        (* End of MultiPortSwitch: '<S729>/Multiport Switch' *)
        

        (* Sum: '<S308>/Add' incorporates:
         *  Constant: '<S304>/Constant'
         *  Product: '<S308>/Product' *)
        rtb_Add_d := USINT_TO_REAL(C_Actia_Batt2_ADS_8[5]) * 5.0;
        (* Sum: '<S547>/Add' incorporates:
         *  ArithShift: '<S546>/Shift Arithmetic'
         *  DataTypeConversion: '<S546>/Data Type Conversion'
         *  Sum: '<S546>/Add' *)
        rtb_Add_ci := DINT_TO_REAL(DWORD_TO_DINT(SHL(DINT_TO_DWORD(USINT_TO_DINT(C_LB_Batt2_InsulationMonitor_Msg[1])), 8)) + USINT_TO_DINT(C_LB_Batt2_InsulationMonitor_Msg[0]));
        (* Switch: '<S547>/Switch' incorporates:
         *  Constant: '<S543>/Constant4' *)

        IF C_LB_Batt2_InsulationMonitor_Timeout THEN 
            rtb_Add_ci := 0.0;
        END_IF;

        (* End of Switch: '<S547>/Switch' *)
        

        (* Sum: '<S730>/Subtract' incorporates:
         *  Constant: '<S730>/Constant4'
         *  Gain: '<S730>/mV to V' *)
        rtb_Add_ci := (0.001 * rtb_Add_ci) - 2.48;
        (* MultiPortSwitch: '<S727>/Multiport Switch' incorporates:
         *  Abs: '<S730>/Abs'
         *  Constant: '<S727>/Constant'
         *  Constant: '<S730>/Constant1'
         *  Constant: '<S730>/Constant2'
         *  Product: '<S730>/Divide'
         *  Product: '<S730>/Product'
         *  Sum: '<S730>/Subtract1' *)

        CASE TRUNC(rtb_BattSelect) OF
            1: 
                (* Switch: '<S308>/Switch' incorporates:
                 *  Constant: '<S304>/Constant3'
                 *  Constant: '<S304>/SafeValue_NA '
                 *  RelationalOperator: '<S308>/GreaterThan'
                 *  Switch: '<S308>/Switch1' *)

                IF C_Actia_Batt2_ADS_8_Timeout THEN 
                    rtb_Add_d := 0.0;
                ELSIF rtb_Add_d > 0.0 THEN 
                    (* Switch: '<S308>/Switch1' incorporates:
                     *  Constant: '<S304>/SafeValue_Error' *)
                    rtb_Add_d := 0.0;
                END_IF;

                (* End of Switch: '<S308>/Switch' *)
            2: 
                rtb_Add_d := ((rtb_Add_ic * 10.0) / ABS(rtb_Add_ci)) - 2000.0;
            3: 
                rtb_Add_d := 0.0;
            ELSE
                rtb_Add_d := 0.0;
        END_CASE;

        (* End of MultiPortSwitch: '<S727>/Multiport Switch' *)
        

        (* Sum: '<S369>/Add' incorporates:
         *  Constant: '<S365>/Constant'
         *  Product: '<S369>/Product' *)
        rtb_Add_ky := USINT_TO_REAL(C_Actia_Batt3_ADS_8[5]) * 5.0;
        (* Sum: '<S627>/Add' incorporates:
         *  ArithShift: '<S626>/Shift Arithmetic'
         *  DataTypeConversion: '<S626>/Data Type Conversion'
         *  Sum: '<S626>/Add' *)
        rtb_Add_ci := DINT_TO_REAL(DWORD_TO_DINT(SHL(DINT_TO_DWORD(USINT_TO_DINT(C_LB_Batt3_InsulationMonitor_Msg[1])), 8)) + USINT_TO_DINT(C_LB_Batt3_InsulationMonitor_Msg[0]));
        (* Switch: '<S627>/Switch' incorporates:
         *  Constant: '<S623>/Constant4' *)

        IF C_LB_Batt3_InsulationMonitor_Timeout THEN 
            rtb_Add_ci := 0.0;
        END_IF;

        (* End of Switch: '<S627>/Switch' *)
        

        (* Sum: '<S731>/Subtract' incorporates:
         *  Constant: '<S731>/Constant4'
         *  Gain: '<S731>/mV to V' *)
        rtb_Add_ci := (0.001 * rtb_Add_ci) - 2.48;
        (* MultiPortSwitch: '<S728>/Multiport Switch' incorporates:
         *  Abs: '<S731>/Abs'
         *  Constant: '<S728>/Constant'
         *  Constant: '<S731>/Constant1'
         *  Constant: '<S731>/Constant2'
         *  Product: '<S731>/Divide'
         *  Product: '<S731>/Product'
         *  Sum: '<S731>/Subtract1' *)

        CASE TRUNC(rtb_BattSelect_i) OF
            1: 
                (* Switch: '<S369>/Switch' incorporates:
                 *  Constant: '<S365>/Constant3'
                 *  Constant: '<S365>/SafeValue_NA '
                 *  RelationalOperator: '<S369>/GreaterThan'
                 *  Switch: '<S369>/Switch1' *)

                IF C_Actia_Batt3_ADS_8_Timeout THEN 
                    rtb_Add_ky := 0.0;
                ELSIF rtb_Add_ky > 0.0 THEN 
                    (* Switch: '<S369>/Switch1' incorporates:
                     *  Constant: '<S365>/SafeValue_Error' *)
                    rtb_Add_ky := 0.0;
                END_IF;

                (* End of Switch: '<S369>/Switch' *)
            2: 
                rtb_Add_ky := ((rtb_Add_en * 10.0) / ABS(rtb_Add_ci)) - 2000.0;
            3: 
                rtb_Add_ky := 0.0;
            ELSE
                rtb_Add_ky := 0.0;
        END_CASE;

        (* End of MultiPortSwitch: '<S728>/Multiport Switch' *)
        

        (* Sum: '<S469>/Add' incorporates:
         *  ArithShift: '<S468>/Shift Arithmetic'
         *  DataTypeConversion: '<S468>/Data Type Conversion'
         *  Sum: '<S468>/Add' *)
        rtb_Add_ci := DINT_TO_REAL(DWORD_TO_DINT(SHL(DINT_TO_DWORD(USINT_TO_DINT(C_LB_Batt1_InsulationMonitor_Msg[3])), 8)) + USINT_TO_DINT(C_LB_Batt1_InsulationMonitor_Msg[2]));
        (* Switch: '<S469>/Switch' incorporates:
         *  Constant: '<S464>/Constant4' *)

        IF C_LB_Batt1_InsulationMonitor_Timeout THEN 
            rtb_Add_ci := 0.0;
        END_IF;

        (* End of Switch: '<S469>/Switch' *)
        

        (* Sum: '<S732>/Subtract3' incorporates:
         *  Abs: '<S732>/Abs1'
         *  Constant: '<S732>/Constant5'
         *  Constant: '<S732>/Constant6'
         *  Constant: '<S732>/Constant7'
         *  Gain: '<S732>/mV to V1'
         *  Product: '<S732>/Divide1'
         *  Product: '<S732>/Product1'
         *  Sum: '<S732>/Subtract2' *)
        rtb_Add_psl := ((rtb_Add_psl * 10.0) / ABS((0.001 * rtb_Add_ci) - 2.48)) - 2000.0;
        (* Sum: '<S549>/Add' incorporates:
         *  ArithShift: '<S548>/Shift Arithmetic'
         *  DataTypeConversion: '<S548>/Data Type Conversion'
         *  Sum: '<S548>/Add' *)
        rtb_Add_ci := DINT_TO_REAL(DWORD_TO_DINT(SHL(DINT_TO_DWORD(USINT_TO_DINT(C_LB_Batt2_InsulationMonitor_Msg[3])), 8)) + USINT_TO_DINT(C_LB_Batt2_InsulationMonitor_Msg[2]));
        (* Switch: '<S549>/Switch' incorporates:
         *  Constant: '<S544>/Constant4' *)

        IF C_LB_Batt2_InsulationMonitor_Timeout THEN 
            rtb_Add_ci := 0.0;
        END_IF;

        (* End of Switch: '<S549>/Switch' *)
        

        (* Sum: '<S730>/Subtract3' incorporates:
         *  Abs: '<S730>/Abs1'
         *  Constant: '<S730>/Constant5'
         *  Constant: '<S730>/Constant6'
         *  Constant: '<S730>/Constant7'
         *  Gain: '<S730>/mV to V1'
         *  Product: '<S730>/Divide1'
         *  Product: '<S730>/Product1'
         *  Sum: '<S730>/Subtract2' *)
        rtb_Add_ic := ((rtb_Add_ic * 10.0) / ABS((0.001 * rtb_Add_ci) - 2.48)) - 2000.0;
        (* Sum: '<S629>/Add' incorporates:
         *  ArithShift: '<S628>/Shift Arithmetic'
         *  DataTypeConversion: '<S628>/Data Type Conversion'
         *  Sum: '<S628>/Add' *)
        rtb_Add_ci := DINT_TO_REAL(DWORD_TO_DINT(SHL(DINT_TO_DWORD(USINT_TO_DINT(C_LB_Batt3_InsulationMonitor_Msg[3])), 8)) + USINT_TO_DINT(C_LB_Batt3_InsulationMonitor_Msg[2]));
        (* Switch: '<S629>/Switch' incorporates:
         *  Constant: '<S624>/Constant4' *)

        IF C_LB_Batt3_InsulationMonitor_Timeout THEN 
            rtb_Add_ci := 0.0;
        END_IF;

        (* End of Switch: '<S629>/Switch' *)
        

        (* Sum: '<S731>/Subtract3' incorporates:
         *  Abs: '<S731>/Abs1'
         *  Constant: '<S731>/Constant5'
         *  Constant: '<S731>/Constant6'
         *  Constant: '<S731>/Constant7'
         *  Gain: '<S731>/mV to V1'
         *  Product: '<S731>/Divide1'
         *  Product: '<S731>/Product1'
         *  Sum: '<S731>/Subtract2' *)
        rtb_Add_en := ((rtb_Add_en * 10.0) / ABS((0.001 * rtb_Add_ci) - 2.48)) - 2000.0;
        (* Sum: '<S259>/Add' incorporates:
         *  Product: '<S259>/Product' *)
        rtb_Switch_a := USINT_TO_REAL(C_Actia_Batt1_ADS_1[7]);
        (* MultiPortSwitch: '<S726>/Multiport Switch' incorporates:
         *  Constant: '<S726>/Constant'
         *  Constant: '<S726>/Constant1' *)

        CASE TRUNC(rtb_BattSelect_f) OF
            1: 
                (* Switch: '<S259>/Switch' incorporates:
                 *  Constant: '<S254>/SafeValue_NA ' *)

                IF C_Actia_Batt1_ADS_1_Timeout THEN 
                    rtb_Switch_a := 0.0;
                END_IF;

                (* End of Switch: '<S259>/Switch' *)
            2: 
                rtb_Switch_a := 25.0;
            3: 
                rtb_Switch_a := 0.0;
            ELSE
                rtb_Switch_a := 0.0;
        END_CASE;

        (* End of MultiPortSwitch: '<S726>/Multiport Switch' *)
        

        (* Sum: '<S318>/Add' incorporates:
         *  Product: '<S318>/Product' *)
        rtb_Add_c0 := USINT_TO_REAL(C_Actia_Batt2_ADS_1[7]);
        (* MultiPortSwitch: '<S724>/Multiport Switch' incorporates:
         *  Constant: '<S724>/Constant'
         *  Constant: '<S724>/Constant1' *)

        CASE TRUNC(rtb_BattSelect) OF
            1: 
                (* Switch: '<S318>/Switch' incorporates:
                 *  Constant: '<S314>/SafeValue_NA ' *)

                IF C_Actia_Batt2_ADS_1_Timeout THEN 
                    rtb_Add_c0 := 0.0;
                END_IF;

                (* End of Switch: '<S318>/Switch' *)
            2: 
                rtb_Add_c0 := 25.0;
            3: 
                rtb_Add_c0 := 0.0;
            ELSE
                rtb_Add_c0 := 0.0;
        END_CASE;

        (* End of MultiPortSwitch: '<S724>/Multiport Switch' *)
        

        (* Sum: '<S381>/Add' incorporates:
         *  Product: '<S381>/Product' *)
        rtb_Add_egs := USINT_TO_REAL(C_Actia_Batt3_ADS_1[7]);
        (* MultiPortSwitch: '<S725>/Multiport Switch' incorporates:
         *  Constant: '<S725>/Constant'
         *  Constant: '<S725>/Constant1' *)

        CASE TRUNC(rtb_BattSelect_i) OF
            1: 
                (* Switch: '<S381>/Switch' incorporates:
                 *  Constant: '<S376>/SafeValue_NA ' *)

                IF C_Actia_Batt3_ADS_1_Timeout THEN 
                    rtb_Add_egs := 0.0;
                END_IF;

                (* End of Switch: '<S381>/Switch' *)
            2: 
                rtb_Add_egs := 25.0;
            3: 
                rtb_Add_egs := 0.0;
            ELSE
                rtb_Add_egs := 0.0;
        END_CASE;

        (* End of MultiPortSwitch: '<S725>/Multiport Switch' *)
        

        (* Outputs for Enabled SubSystem: '<S203>/Subsystem' incorporates:
         *  EnablePort: '<S232>/Timeout' *)
        (* Logic: '<S203>/NOT' *)

        IF  NOT C_Actia_Batt1_Error_Timeout THEN 

            IF  NOT Subsystem_MODE_h THEN 
                Subsystem_MODE_h := TRUE;
            END_IF;

            (* DataTypeConversion: '<S232>/Data Type Conversion2' incorporates:
             *  DataTypeConversion: '<S235>/Extract Desired Bits' *)
            IP_boBatt1_HV_relay_PLUS_Sense := DWORD_TO_UDINT(UDINT_TO_DWORD(USINT_TO_UDINT(C_Actia_Batt1_Error[6])) AND 1) <> 0;
            (* DataTypeConversion: '<S232>/Data Type Conversion4' incorporates:
             *  DataTypeConversion: '<S237>/Extract Desired Bits' *)
            IP_boBatt1_HV_relay_MINUS_Sense := DWORD_TO_UDINT(UDINT_TO_DWORD(DINT_TO_UDINT(DWORD_TO_DINT(SHR(DINT_TO_DWORD(USINT_TO_DINT(C_Actia_Batt1_Error[6])), 2)))) AND 1) <> 0;
            (* DataTypeConversion: '<S232>/Data Type Conversion5' incorporates:
             *  DataTypeConversion: '<S238>/Extract Desired Bits' *)
            IP_boBatt1_IMD_active := DWORD_TO_UDINT(UDINT_TO_DWORD(DINT_TO_UDINT(DWORD_TO_DINT(SHR(DINT_TO_DWORD(USINT_TO_DINT(C_Actia_Batt1_Error[6])), 4)))) AND 1) <> 0;
        ELSIF Subsystem_MODE_h THEN 
            (* Disable for DataTypeConversion: '<S232>/Data Type Conversion2' incorporates:
             *  Outport: '<S232>/IP_boBatt1_HV_relay_PLUS_Sense' *)
            IP_boBatt1_HV_relay_PLUS_Sense := FALSE;
            (* Disable for DataTypeConversion: '<S232>/Data Type Conversion4' incorporates:
             *  Outport: '<S232>/IP_boBatt1_HV_relay_MINUS_Sense' *)
            IP_boBatt1_HV_relay_MINUS_Sense := FALSE;
            (* Disable for DataTypeConversion: '<S232>/Data Type Conversion5' incorporates:
             *  Outport: '<S232>/IP_boBatt1_IMD_active' *)
            IP_boBatt1_IMD_active := FALSE;
            Subsystem_MODE_h := FALSE;
        END_IF;

        (* End of Logic: '<S203>/NOT' *)
        (* End of Outputs for SubSystem: '<S203>/Subsystem' *)
        

        (* MultiPortSwitch: '<S780>/Multiport Switch' incorporates:
         *  Constant: '<S780>/Constant'
         *  Constant: '<S796>/Constant'
         *  Constant: '<S797>/Constant'
         *  Constant: '<S798>/Constant'
         *  Logic: '<S780>/OR'
         *  RelationalOperator: '<S796>/Compare'
         *  RelationalOperator: '<S797>/Compare'
         *  RelationalOperator: '<S798>/Compare' *)

        CASE TRUNC(rtb_BattSelect_f) OF
            1: 
                rtb_IP_boBMS_HV_Minus_Sense_BB1 := IP_boBatt1_HV_relay_MINUS_Sense;
                (* MultiPortSwitch: '<S775>/Multiport Switch' *)
                rtb_IP_boBMS_HV_Plus_Sense_BB1 := IP_boBatt1_HV_relay_PLUS_Sense;
            2: 
                rtb_IP_boBMS_HV_Minus_Sense_BB1 := ((rtb_Add_nm = 64.0) OR (rtb_Add_nm = 96.0)) OR (rtb_Add_nm = 224.0);
                (* MultiPortSwitch: '<S775>/Multiport Switch' incorporates:
                 *  Constant: '<S781>/Constant'
                 *  Constant: '<S782>/Constant'
                 *  Constant: '<S783>/Constant'
                 *  Constant: '<S796>/Constant'
                 *  Constant: '<S797>/Constant'
                 *  Constant: '<S798>/Constant'
                 *  Logic: '<S775>/OR'
                 *  Logic: '<S780>/OR'
                 *  RelationalOperator: '<S781>/Compare'
                 *  RelationalOperator: '<S782>/Compare'
                 *  RelationalOperator: '<S783>/Compare'
                 *  RelationalOperator: '<S796>/Compare'
                 *  RelationalOperator: '<S797>/Compare'
                 *  RelationalOperator: '<S798>/Compare' *)
                rtb_IP_boBMS_HV_Plus_Sense_BB1 := ((rtb_Add_nm = 128.0) OR (rtb_Add_nm = 160.0)) OR (rtb_Add_nm = 224.0);
            3: 
                rtb_IP_boBMS_HV_Minus_Sense_BB1 := FALSE;
                (* MultiPortSwitch: '<S775>/Multiport Switch' incorporates:
                 *  Constant: '<S775>/Constant'
                 *  Constant: '<S780>/Constant' *)
                rtb_IP_boBMS_HV_Plus_Sense_BB1 := FALSE;
            ELSE
                rtb_IP_boBMS_HV_Minus_Sense_BB1 := FALSE;
                (* MultiPortSwitch: '<S775>/Multiport Switch' incorporates:
                 *  Constant: '<S775>/Constant'
                 *  Constant: '<S780>/Constant' *)
                rtb_IP_boBMS_HV_Plus_Sense_BB1 := FALSE;
        END_CASE;

        (* End of MultiPortSwitch: '<S780>/Multiport Switch' *)
        

        (* Outputs for Enabled SubSystem: '<S264>/Subsystem' incorporates:
         *  EnablePort: '<S293>/Timeout' *)
        (* Logic: '<S264>/NOT' *)

        IF  NOT C_Actia_Batt2_Error_Timeout THEN 

            IF  NOT Subsystem_MODE_c THEN 
                Subsystem_MODE_c := TRUE;
            END_IF;

            (* DataTypeConversion: '<S293>/Data Type Conversion2' incorporates:
             *  DataTypeConversion: '<S296>/Extract Desired Bits' *)
            IP_boBatt2_HV_relay_PLUS_Sense := DWORD_TO_UDINT(UDINT_TO_DWORD(USINT_TO_UDINT(C_Actia_Batt2_Error[6])) AND 1) <> 0;
            (* DataTypeConversion: '<S293>/Data Type Conversion4' incorporates:
             *  DataTypeConversion: '<S298>/Extract Desired Bits' *)
            IP_boBatt2_HV_relay_MINUS_Sense := DWORD_TO_UDINT(UDINT_TO_DWORD(DINT_TO_UDINT(DWORD_TO_DINT(SHR(DINT_TO_DWORD(USINT_TO_DINT(C_Actia_Batt2_Error[6])), 2)))) AND 1) <> 0;
            (* DataTypeConversion: '<S293>/Data Type Conversion5' incorporates:
             *  DataTypeConversion: '<S299>/Extract Desired Bits' *)
            IP_boBatt2_IMD_active := DWORD_TO_UDINT(UDINT_TO_DWORD(DINT_TO_UDINT(DWORD_TO_DINT(SHR(DINT_TO_DWORD(USINT_TO_DINT(C_Actia_Batt2_Error[6])), 4)))) AND 1) <> 0;
        ELSIF Subsystem_MODE_c THEN 
            (* Disable for DataTypeConversion: '<S293>/Data Type Conversion2' incorporates:
             *  Outport: '<S293>/IP_boBatt2_HV_relay_PLUS_Sense' *)
            IP_boBatt2_HV_relay_PLUS_Sense := FALSE;
            (* Disable for DataTypeConversion: '<S293>/Data Type Conversion4' incorporates:
             *  Outport: '<S293>/IP_boBatt2_HV_relay_MINUS_Sense' *)
            IP_boBatt2_HV_relay_MINUS_Sense := FALSE;
            (* Disable for DataTypeConversion: '<S293>/Data Type Conversion5' incorporates:
             *  Outport: '<S293>/IP_boBatt2_IMD_active' *)
            IP_boBatt2_IMD_active := FALSE;
            Subsystem_MODE_c := FALSE;
        END_IF;

        (* End of Logic: '<S264>/NOT' *)
        (* End of Outputs for SubSystem: '<S264>/Subsystem' *)
        

        (* MultiPortSwitch: '<S777>/Multiport Switch' incorporates:
         *  Constant: '<S777>/Constant'
         *  Constant: '<S787>/Constant'
         *  Constant: '<S788>/Constant'
         *  Constant: '<S789>/Constant'
         *  Logic: '<S777>/OR'
         *  RelationalOperator: '<S787>/Compare'
         *  RelationalOperator: '<S788>/Compare'
         *  RelationalOperator: '<S789>/Compare' *)

        CASE TRUNC(rtb_BattSelect) OF
            1: 
                rtb_IP_boBMS_HV_Minus_Sense_BB2 := IP_boBatt2_HV_relay_MINUS_Sense;
                (* MultiPortSwitch: '<S776>/Multiport Switch' *)
                rtb_IP_boBMS_HV_Plus_Sense_BB2 := IP_boBatt2_HV_relay_PLUS_Sense;
            2: 
                rtb_IP_boBMS_HV_Minus_Sense_BB2 := ((rtb_Add_d4 = 64.0) OR (rtb_Add_d4 = 96.0)) OR (rtb_Add_d4 = 224.0);
                (* MultiPortSwitch: '<S776>/Multiport Switch' incorporates:
                 *  Constant: '<S784>/Constant'
                 *  Constant: '<S785>/Constant'
                 *  Constant: '<S786>/Constant'
                 *  Constant: '<S787>/Constant'
                 *  Constant: '<S788>/Constant'
                 *  Constant: '<S789>/Constant'
                 *  Logic: '<S776>/OR'
                 *  Logic: '<S777>/OR'
                 *  RelationalOperator: '<S784>/Compare'
                 *  RelationalOperator: '<S785>/Compare'
                 *  RelationalOperator: '<S786>/Compare'
                 *  RelationalOperator: '<S787>/Compare'
                 *  RelationalOperator: '<S788>/Compare'
                 *  RelationalOperator: '<S789>/Compare' *)
                rtb_IP_boBMS_HV_Plus_Sense_BB2 := ((rtb_Add_d4 = 128.0) OR (rtb_Add_d4 = 160.0)) OR (rtb_Add_d4 = 224.0);
            3: 
                rtb_IP_boBMS_HV_Minus_Sense_BB2 := FALSE;
                (* MultiPortSwitch: '<S776>/Multiport Switch' incorporates:
                 *  Constant: '<S776>/Constant'
                 *  Constant: '<S777>/Constant' *)
                rtb_IP_boBMS_HV_Plus_Sense_BB2 := FALSE;
            ELSE
                rtb_IP_boBMS_HV_Minus_Sense_BB2 := FALSE;
                (* MultiPortSwitch: '<S776>/Multiport Switch' incorporates:
                 *  Constant: '<S776>/Constant'
                 *  Constant: '<S777>/Constant' *)
                rtb_IP_boBMS_HV_Plus_Sense_BB2 := FALSE;
        END_CASE;

        (* End of MultiPortSwitch: '<S777>/Multiport Switch' *)
        

        (* Outputs for Enabled SubSystem: '<S325>/Subsystem' incorporates:
         *  EnablePort: '<S354>/Timeout' *)
        (* Logic: '<S325>/NOT' *)

        IF  NOT C_Actia_Batt3_Error_Timeout THEN 

            IF  NOT Subsystem_MODE THEN 
                Subsystem_MODE := TRUE;
            END_IF;

            (* DataTypeConversion: '<S354>/Data Type Conversion2' incorporates:
             *  DataTypeConversion: '<S357>/Extract Desired Bits' *)
            IP_boBatt3_HV_relay_PLUS_Sense := DWORD_TO_UDINT(UDINT_TO_DWORD(USINT_TO_UDINT(C_Actia_Batt3_Error[6])) AND 1) <> 0;
            (* DataTypeConversion: '<S354>/Data Type Conversion4' incorporates:
             *  DataTypeConversion: '<S359>/Extract Desired Bits' *)
            IP_boBatt3_HV_relay_MINUS_Sense := DWORD_TO_UDINT(UDINT_TO_DWORD(DINT_TO_UDINT(DWORD_TO_DINT(SHR(DINT_TO_DWORD(USINT_TO_DINT(C_Actia_Batt3_Error[6])), 2)))) AND 1) <> 0;
            (* DataTypeConversion: '<S354>/Data Type Conversion5' incorporates:
             *  DataTypeConversion: '<S360>/Extract Desired Bits' *)
            IP_boBatt3_IMD_active := DWORD_TO_UDINT(UDINT_TO_DWORD(DINT_TO_UDINT(DWORD_TO_DINT(SHR(DINT_TO_DWORD(USINT_TO_DINT(C_Actia_Batt3_Error[6])), 4)))) AND 1) <> 0;
        ELSIF Subsystem_MODE THEN 
            (* Disable for DataTypeConversion: '<S354>/Data Type Conversion2' incorporates:
             *  Outport: '<S354>/IP_boBatt3_HV_relay_PLUS_Sense' *)
            IP_boBatt3_HV_relay_PLUS_Sense := FALSE;
            (* Disable for DataTypeConversion: '<S354>/Data Type Conversion4' incorporates:
             *  Outport: '<S354>/IP_boBatt3_HV_relay_MINUS_Sense' *)
            IP_boBatt3_HV_relay_MINUS_Sense := FALSE;
            (* Disable for DataTypeConversion: '<S354>/Data Type Conversion5' incorporates:
             *  Outport: '<S354>/IP_boBatt3_IMD_active' *)
            IP_boBatt3_IMD_active := FALSE;
            Subsystem_MODE := FALSE;
        END_IF;

        (* End of Logic: '<S325>/NOT' *)
        (* End of Outputs for SubSystem: '<S325>/Subsystem' *)
        

        (* MultiPortSwitch: '<S779>/Multiport Switch' incorporates:
         *  Constant: '<S779>/Constant'
         *  Constant: '<S793>/Constant'
         *  Constant: '<S794>/Constant'
         *  Constant: '<S795>/Constant'
         *  Logic: '<S779>/OR'
         *  RelationalOperator: '<S793>/Compare'
         *  RelationalOperator: '<S794>/Compare'
         *  RelationalOperator: '<S795>/Compare' *)

        CASE TRUNC(rtb_BattSelect_i) OF
            1: 
                rtb_IP_boBMS_HV_Minus_Sense_BB3 := IP_boBatt3_HV_relay_MINUS_Sense;
                (* MultiPortSwitch: '<S778>/Multiport Switch' *)
                rtb_IP_boBMS_HV_Plus_Sense_BB3 := IP_boBatt3_HV_relay_PLUS_Sense;
            2: 
                rtb_IP_boBMS_HV_Minus_Sense_BB3 := ((rtb_Add_cw = 64.0) OR (rtb_Add_cw = 96.0)) OR (rtb_Add_cw = 224.0);
                (* MultiPortSwitch: '<S778>/Multiport Switch' incorporates:
                 *  Constant: '<S790>/Constant'
                 *  Constant: '<S791>/Constant'
                 *  Constant: '<S792>/Constant'
                 *  Constant: '<S793>/Constant'
                 *  Constant: '<S794>/Constant'
                 *  Constant: '<S795>/Constant'
                 *  Logic: '<S778>/OR'
                 *  Logic: '<S779>/OR'
                 *  RelationalOperator: '<S790>/Compare'
                 *  RelationalOperator: '<S791>/Compare'
                 *  RelationalOperator: '<S792>/Compare'
                 *  RelationalOperator: '<S793>/Compare'
                 *  RelationalOperator: '<S794>/Compare'
                 *  RelationalOperator: '<S795>/Compare' *)
                rtb_IP_boBMS_HV_Plus_Sense_BB3 := ((rtb_Add_cw = 128.0) OR (rtb_Add_cw = 160.0)) OR (rtb_Add_cw = 224.0);
            3: 
                rtb_IP_boBMS_HV_Minus_Sense_BB3 := FALSE;
                (* MultiPortSwitch: '<S778>/Multiport Switch' incorporates:
                 *  Constant: '<S778>/Constant'
                 *  Constant: '<S779>/Constant' *)
                rtb_IP_boBMS_HV_Plus_Sense_BB3 := FALSE;
            ELSE
                rtb_IP_boBMS_HV_Minus_Sense_BB3 := FALSE;
                (* MultiPortSwitch: '<S778>/Multiport Switch' incorporates:
                 *  Constant: '<S778>/Constant'
                 *  Constant: '<S779>/Constant' *)
                rtb_IP_boBMS_HV_Plus_Sense_BB3 := FALSE;
        END_CASE;

        (* End of MultiPortSwitch: '<S779>/Multiport Switch' *)
        

        (* Delay: '<S768>/Delay' incorporates:
         *  Constant: '<S768>/Constant1' *)
        i2_IMD_OK(ssMethodType := SS_OUTPUT, IP_boBMS_InsulationReadyOK := DI_IMD_FB_BB1, Req_IMD := Delay_DSTATE[0], IT_u8IMD_DelayTime_s_g := IT_u8IMD_DelayTime_s);
        rtb_S_in := i2_IMD_OK.IMD_OK_i;
        (* MultiPortSwitch: '<S768>/Multiport Switch' incorporates:
         *  Constant: '<S768>/Constant' *)

        CASE TRUNC(rtb_BattSelect_f) OF
            1: 
                rtb_S_in := IP_boBatt1_Insulation_ready_and_OK;
            2: 
                ;
                ;
            3: 
                rtb_S_in := FALSE;
            ELSE
                rtb_S_in := FALSE;
        END_CASE;

        (* End of MultiPortSwitch: '<S768>/Multiport Switch' *)
        

        (* Delay: '<S766>/Delay' incorporates:
         *  Constant: '<S766>/Constant1' *)
        i0_IMD_OK(ssMethodType := SS_OUTPUT, IP_boBMS_InsulationReadyOK := DI_IMD_FB_BB2, Req_IMD := Delay_DSTATE_o[0], IT_u8IMD_DelayTime_s_g := IT_u8IMD_DelayTime_s);
        rtb_IP_boBatt1_Actia_Availability := i0_IMD_OK.IMD_OK_i;
        (* MultiPortSwitch: '<S766>/Multiport Switch' incorporates:
         *  Constant: '<S766>/Constant' *)

        CASE TRUNC(rtb_BattSelect) OF
            1: 
                rtb_IP_boBatt1_Actia_Availability := IP_boBatt2_Insulation_ready_and_OK;
            2: 
                ;
                ;
            3: 
                rtb_IP_boBatt1_Actia_Availability := FALSE;
            ELSE
                rtb_IP_boBatt1_Actia_Availability := FALSE;
        END_CASE;

        (* End of MultiPortSwitch: '<S766>/Multiport Switch' *)
        

        (* Delay: '<S767>/Delay' incorporates:
         *  Constant: '<S767>/Constant1' *)
        i1_IMD_OK(ssMethodType := SS_OUTPUT, IP_boBMS_InsulationReadyOK := DI_IMD_FB_BB3, Req_IMD := Delay_DSTATE_k[0], IT_u8IMD_DelayTime_s_g := IT_u8IMD_DelayTime_s);
        rtb_Delay_dl := i1_IMD_OK.IMD_OK_i;
        (* MultiPortSwitch: '<S767>/Multiport Switch' incorporates:
         *  Constant: '<S767>/Constant' *)

        CASE TRUNC(rtb_BattSelect_i) OF
            1: 
                rtb_Delay_dl := IP_boBatt3_Insulation_ready_and_OK;
            2: 
                ;
                ;
            3: 
                rtb_Delay_dl := FALSE;
            ELSE
                rtb_Delay_dl := FALSE;
        END_CASE;

        (* End of MultiPortSwitch: '<S767>/Multiport Switch' *)
        

        (* Sum: '<S229>/Add' incorporates:
         *  ArithShift: '<S228>/Shift Arithmetic'
         *  DataTypeConversion: '<S228>/Data Type Conversion'
         *  Sum: '<S228>/Add' *)
        rtb_Add_nm := DINT_TO_REAL(DWORD_TO_DINT(SHL(DINT_TO_DWORD(USINT_TO_DINT(C_Actia_Batt1_ADS_0[4])), 8)) + USINT_TO_DINT(C_Actia_Batt1_ADS_0[3]));
        (* Sum: '<S450>/Add' incorporates:
         *  ArithShift: '<S449>/Shift Arithmetic'
         *  Constant: '<S446>/Constant'
         *  DataTypeConversion: '<S449>/Data Type Conversion'
         *  Product: '<S450>/Product'
         *  Sum: '<S449>/Add' *)
        rtb_Add_d4 := DINT_TO_REAL(DWORD_TO_DINT(SHL(DINT_TO_DWORD(USINT_TO_DINT(C_LB_Batt1_CellVoltage01_Msg[1])), 8)) + USINT_TO_DINT(C_LB_Batt1_CellVoltage01_Msg[0])) * 0.1;
        (* MultiPortSwitch: '<S735>/Multiport Switch' incorporates:
         *  Constant: '<S735>/Constant' *)

        CASE TRUNC(rtb_BattSelect_f) OF
            1: 
                (* Switch: '<S229>/Switch' incorporates:
                 *  Constant: '<S226>/Constant7'
                 *  Constant: '<S226>/Constant9'
                 *  RelationalOperator: '<S229>/GreaterThan'
                 *  Switch: '<S229>/Switch1' *)

                IF C_Actia_Batt1_ADS_0_Timeout THEN 
                    rtb_Add_nm := 0.0;
                ELSIF rtb_Add_nm > 4500.0 THEN 
                    (* Switch: '<S229>/Switch1' incorporates:
                     *  Constant: '<S226>/Constant8' *)
                    rtb_Add_nm := 0.0;
                END_IF;

                (* End of Switch: '<S229>/Switch' *)
            2: 
                (* Switch: '<S450>/Switch' incorporates:
                 *  Constant: '<S446>/Constant3'
                 *  Constant: '<S446>/Constant4'
                 *  RelationalOperator: '<S450>/GreaterThan'
                 *  Switch: '<S450>/Switch1' *)

                IF C_LB_Batt1_CellVoltage01_Timeout THEN 
                    rtb_Add_nm := 0.0;
                ELSIF rtb_Add_d4 > 6553.5 THEN 
                    (* Switch: '<S450>/Switch1' incorporates:
                     *  Constant: '<S446>/Constant4' *)
                    rtb_Add_nm := 0.0;
                ELSE 
                    (* Switch: '<S450>/Switch1' *)
                    rtb_Add_nm := rtb_Add_d4;
                END_IF;

                (* End of Switch: '<S450>/Switch' *)
            3: 
                rtb_Add_nm := 0.0;
            ELSE
                rtb_Add_nm := 0.0;
        END_CASE;

        (* End of MultiPortSwitch: '<S735>/Multiport Switch' *)
        

        (* Sum: '<S290>/Add' incorporates:
         *  ArithShift: '<S289>/Shift Arithmetic'
         *  DataTypeConversion: '<S289>/Data Type Conversion'
         *  Sum: '<S289>/Add' *)
        rtb_Add_d4 := DINT_TO_REAL(DWORD_TO_DINT(SHL(DINT_TO_DWORD(USINT_TO_DINT(C_Actia_Batt2_ADS_0[4])), 8)) + USINT_TO_DINT(C_Actia_Batt2_ADS_0[3]));
        (* Sum: '<S530>/Add' incorporates:
         *  ArithShift: '<S529>/Shift Arithmetic'
         *  Constant: '<S526>/Constant'
         *  DataTypeConversion: '<S529>/Data Type Conversion'
         *  Product: '<S530>/Product'
         *  Sum: '<S529>/Add' *)
        rtb_Add_cw := DINT_TO_REAL(DWORD_TO_DINT(SHL(DINT_TO_DWORD(USINT_TO_DINT(C_LB_Batt2_CellVoltage01_Msg[1])), 8)) + USINT_TO_DINT(C_LB_Batt2_CellVoltage01_Msg[0])) * 0.1;
        (* MultiPortSwitch: '<S733>/Multiport Switch' incorporates:
         *  Constant: '<S733>/Constant' *)

        CASE TRUNC(rtb_BattSelect) OF
            1: 
                (* Switch: '<S290>/Switch' incorporates:
                 *  Constant: '<S287>/Constant7'
                 *  Constant: '<S287>/Constant9'
                 *  RelationalOperator: '<S290>/GreaterThan'
                 *  Switch: '<S290>/Switch1' *)

                IF C_Actia_Batt2_ADS_0_Timeout THEN 
                    rtb_Add_d4 := 0.0;
                ELSIF rtb_Add_d4 > 4500.0 THEN 
                    (* Switch: '<S290>/Switch1' incorporates:
                     *  Constant: '<S287>/Constant8' *)
                    rtb_Add_d4 := 0.0;
                END_IF;

                (* End of Switch: '<S290>/Switch' *)
            2: 
                (* Switch: '<S530>/Switch' incorporates:
                 *  Constant: '<S526>/Constant3'
                 *  Constant: '<S526>/Constant4'
                 *  RelationalOperator: '<S530>/GreaterThan'
                 *  Switch: '<S530>/Switch1' *)

                IF C_LB_Batt2_CellVoltage01_Timeout THEN 
                    rtb_Add_d4 := 0.0;
                ELSIF rtb_Add_cw > 6553.5 THEN 
                    (* Switch: '<S530>/Switch1' incorporates:
                     *  Constant: '<S526>/Constant4' *)
                    rtb_Add_d4 := 0.0;
                ELSE 
                    (* Switch: '<S530>/Switch1' *)
                    rtb_Add_d4 := rtb_Add_cw;
                END_IF;

                (* End of Switch: '<S530>/Switch' *)
            3: 
                rtb_Add_d4 := 0.0;
            ELSE
                rtb_Add_d4 := 0.0;
        END_CASE;

        (* End of MultiPortSwitch: '<S733>/Multiport Switch' *)
        

        (* Sum: '<S351>/Add' incorporates:
         *  ArithShift: '<S350>/Shift Arithmetic'
         *  DataTypeConversion: '<S350>/Data Type Conversion'
         *  Sum: '<S350>/Add' *)
        rtb_Add_cw := DINT_TO_REAL(DWORD_TO_DINT(SHL(DINT_TO_DWORD(USINT_TO_DINT(C_Actia_Batt3_ADS_0[4])), 8)) + USINT_TO_DINT(C_Actia_Batt3_ADS_0[3]));
        (* Sum: '<S610>/Add' incorporates:
         *  ArithShift: '<S609>/Shift Arithmetic'
         *  Constant: '<S606>/Constant'
         *  DataTypeConversion: '<S609>/Data Type Conversion'
         *  Product: '<S610>/Product'
         *  Sum: '<S609>/Add' *)
        rtb_Add_ie := DINT_TO_REAL(DWORD_TO_DINT(SHL(DINT_TO_DWORD(USINT_TO_DINT(C_LB_Batt3_CellVoltage01_Msg[1])), 8)) + USINT_TO_DINT(C_LB_Batt3_CellVoltage01_Msg[0])) * 0.1;
        (* MultiPortSwitch: '<S734>/Multiport Switch' incorporates:
         *  Constant: '<S734>/Constant' *)

        CASE TRUNC(rtb_BattSelect_i) OF
            1: 
                (* Switch: '<S351>/Switch' incorporates:
                 *  Constant: '<S348>/Constant7'
                 *  Constant: '<S348>/Constant9'
                 *  RelationalOperator: '<S351>/GreaterThan'
                 *  Switch: '<S351>/Switch1' *)

                IF C_Actia_Batt3_ADS_0_Timeout THEN 
                    rtb_Add_cw := 0.0;
                ELSIF rtb_Add_cw > 4500.0 THEN 
                    (* Switch: '<S351>/Switch1' incorporates:
                     *  Constant: '<S348>/Constant8' *)
                    rtb_Add_cw := 0.0;
                END_IF;

                (* End of Switch: '<S351>/Switch' *)
            2: 
                (* Switch: '<S610>/Switch' incorporates:
                 *  Constant: '<S606>/Constant3'
                 *  Constant: '<S606>/Constant4'
                 *  RelationalOperator: '<S610>/GreaterThan'
                 *  Switch: '<S610>/Switch1' *)

                IF C_LB_Batt3_CellVoltage01_Timeout THEN 
                    rtb_Add_cw := 0.0;
                ELSIF rtb_Add_ie > 6553.5 THEN 
                    (* Switch: '<S610>/Switch1' incorporates:
                     *  Constant: '<S606>/Constant4' *)
                    rtb_Add_cw := 0.0;
                ELSE 
                    (* Switch: '<S610>/Switch1' *)
                    rtb_Add_cw := rtb_Add_ie;
                END_IF;

                (* End of Switch: '<S610>/Switch' *)
            3: 
                rtb_Add_cw := 0.0;
            ELSE
                rtb_Add_cw := 0.0;
        END_CASE;

        (* End of MultiPortSwitch: '<S734>/Multiport Switch' *)
        

        (* Sum: '<S231>/Add' incorporates:
         *  ArithShift: '<S230>/Shift Arithmetic'
         *  DataTypeConversion: '<S230>/Data Type Conversion'
         *  Sum: '<S230>/Add' *)
        rtb_Add_ie := DINT_TO_REAL(DWORD_TO_DINT(SHL(DINT_TO_DWORD(USINT_TO_DINT(C_Actia_Batt1_ADS_0[6])), 8)) + USINT_TO_DINT(C_Actia_Batt1_ADS_0[5]));
        (* Sum: '<S454>/Add' incorporates:
         *  ArithShift: '<S453>/Shift Arithmetic'
         *  Constant: '<S448>/Constant'
         *  DataTypeConversion: '<S453>/Data Type Conversion'
         *  Product: '<S454>/Product'
         *  Sum: '<S453>/Add' *)
        rtb_Add_oy := DINT_TO_REAL(DWORD_TO_DINT(SHL(DINT_TO_DWORD(USINT_TO_DINT(C_LB_Batt1_CellVoltage01_Msg[5])), 8)) + USINT_TO_DINT(C_LB_Batt1_CellVoltage01_Msg[4])) * 0.1;
        (* MultiPortSwitch: '<S738>/Multiport Switch' incorporates:
         *  Constant: '<S738>/Constant' *)

        CASE TRUNC(rtb_BattSelect_f) OF
            1: 
                (* Switch: '<S231>/Switch' incorporates:
                 *  Constant: '<S227>/Constant7'
                 *  Constant: '<S227>/Constant9'
                 *  RelationalOperator: '<S231>/GreaterThan'
                 *  Switch: '<S231>/Switch1' *)

                IF C_Actia_Batt1_ADS_0_Timeout THEN 
                    rtb_Add_ie := 0.0;
                ELSIF rtb_Add_ie > 4500.0 THEN 
                    (* Switch: '<S231>/Switch1' incorporates:
                     *  Constant: '<S227>/Constant8' *)
                    rtb_Add_ie := 0.0;
                END_IF;

                (* End of Switch: '<S231>/Switch' *)
            2: 
                (* Switch: '<S454>/Switch' incorporates:
                 *  Constant: '<S448>/Constant3'
                 *  Constant: '<S448>/Constant4'
                 *  RelationalOperator: '<S454>/GreaterThan'
                 *  Switch: '<S454>/Switch1' *)

                IF C_LB_Batt1_CellVoltage01_Timeout THEN 
                    rtb_Add_ie := 0.0;
                ELSIF rtb_Add_oy > 6553.5 THEN 
                    (* Switch: '<S454>/Switch1' incorporates:
                     *  Constant: '<S448>/Constant4' *)
                    rtb_Add_ie := 0.0;
                ELSE 
                    (* Switch: '<S454>/Switch1' *)
                    rtb_Add_ie := rtb_Add_oy;
                END_IF;

                (* End of Switch: '<S454>/Switch' *)
            3: 
                rtb_Add_ie := 0.0;
            ELSE
                rtb_Add_ie := 0.0;
        END_CASE;

        (* End of MultiPortSwitch: '<S738>/Multiport Switch' *)
        

        (* Sum: '<S292>/Add' incorporates:
         *  ArithShift: '<S291>/Shift Arithmetic'
         *  DataTypeConversion: '<S291>/Data Type Conversion'
         *  Sum: '<S291>/Add' *)
        rtb_Add_oy := DINT_TO_REAL(DWORD_TO_DINT(SHL(DINT_TO_DWORD(USINT_TO_DINT(C_Actia_Batt2_ADS_0[6])), 8)) + USINT_TO_DINT(C_Actia_Batt2_ADS_0[5]));
        (* Sum: '<S534>/Add' incorporates:
         *  ArithShift: '<S533>/Shift Arithmetic'
         *  Constant: '<S528>/Constant'
         *  DataTypeConversion: '<S533>/Data Type Conversion'
         *  Product: '<S534>/Product'
         *  Sum: '<S533>/Add' *)
        rtb_Add_bh := DINT_TO_REAL(DWORD_TO_DINT(SHL(DINT_TO_DWORD(USINT_TO_DINT(C_LB_Batt2_CellVoltage01_Msg[5])), 8)) + USINT_TO_DINT(C_LB_Batt2_CellVoltage01_Msg[4])) * 0.1;
        (* MultiPortSwitch: '<S736>/Multiport Switch' incorporates:
         *  Constant: '<S736>/Constant' *)

        CASE TRUNC(rtb_BattSelect) OF
            1: 
                (* Switch: '<S292>/Switch' incorporates:
                 *  Constant: '<S288>/Constant7'
                 *  Constant: '<S288>/Constant9'
                 *  RelationalOperator: '<S292>/GreaterThan'
                 *  Switch: '<S292>/Switch1' *)

                IF C_Actia_Batt2_ADS_0_Timeout THEN 
                    rtb_Add_oy := 0.0;
                ELSIF rtb_Add_oy > 4500.0 THEN 
                    (* Switch: '<S292>/Switch1' incorporates:
                     *  Constant: '<S288>/Constant8' *)
                    rtb_Add_oy := 0.0;
                END_IF;

                (* End of Switch: '<S292>/Switch' *)
            2: 
                (* Switch: '<S534>/Switch' incorporates:
                 *  Constant: '<S528>/Constant3'
                 *  Constant: '<S528>/Constant4'
                 *  RelationalOperator: '<S534>/GreaterThan'
                 *  Switch: '<S534>/Switch1' *)

                IF C_LB_Batt2_CellVoltage01_Timeout THEN 
                    rtb_Add_oy := 0.0;
                ELSIF rtb_Add_bh > 6553.5 THEN 
                    (* Switch: '<S534>/Switch1' incorporates:
                     *  Constant: '<S528>/Constant4' *)
                    rtb_Add_oy := 0.0;
                ELSE 
                    (* Switch: '<S534>/Switch1' *)
                    rtb_Add_oy := rtb_Add_bh;
                END_IF;

                (* End of Switch: '<S534>/Switch' *)
            3: 
                rtb_Add_oy := 0.0;
            ELSE
                rtb_Add_oy := 0.0;
        END_CASE;

        (* End of MultiPortSwitch: '<S736>/Multiport Switch' *)
        

        (* Sum: '<S353>/Add' incorporates:
         *  ArithShift: '<S352>/Shift Arithmetic'
         *  DataTypeConversion: '<S352>/Data Type Conversion'
         *  Sum: '<S352>/Add' *)
        rtb_Add_bh := DINT_TO_REAL(DWORD_TO_DINT(SHL(DINT_TO_DWORD(USINT_TO_DINT(C_Actia_Batt3_ADS_0[6])), 8)) + USINT_TO_DINT(C_Actia_Batt3_ADS_0[5]));
        (* Sum: '<S614>/Add' incorporates:
         *  ArithShift: '<S613>/Shift Arithmetic'
         *  Constant: '<S608>/Constant'
         *  DataTypeConversion: '<S613>/Data Type Conversion'
         *  Product: '<S614>/Product'
         *  Sum: '<S613>/Add' *)
        rtb_Add_no := DINT_TO_REAL(DWORD_TO_DINT(SHL(DINT_TO_DWORD(USINT_TO_DINT(C_LB_Batt3_CellVoltage01_Msg[5])), 8)) + USINT_TO_DINT(C_LB_Batt3_CellVoltage01_Msg[4])) * 0.1;
        (* MultiPortSwitch: '<S737>/Multiport Switch' incorporates:
         *  Constant: '<S737>/Constant' *)

        CASE TRUNC(rtb_BattSelect_i) OF
            1: 
                (* Switch: '<S353>/Switch' incorporates:
                 *  Constant: '<S349>/Constant7'
                 *  Constant: '<S349>/Constant9'
                 *  RelationalOperator: '<S353>/GreaterThan'
                 *  Switch: '<S353>/Switch1' *)

                IF C_Actia_Batt3_ADS_0_Timeout THEN 
                    rtb_Add_bh := 0.0;
                ELSIF rtb_Add_bh > 4500.0 THEN 
                    (* Switch: '<S353>/Switch1' incorporates:
                     *  Constant: '<S349>/Constant8' *)
                    rtb_Add_bh := 0.0;
                END_IF;

                (* End of Switch: '<S353>/Switch' *)
            2: 
                (* Switch: '<S614>/Switch' incorporates:
                 *  Constant: '<S608>/Constant3'
                 *  Constant: '<S608>/Constant4'
                 *  RelationalOperator: '<S614>/GreaterThan'
                 *  Switch: '<S614>/Switch1' *)

                IF C_LB_Batt3_CellVoltage01_Timeout THEN 
                    rtb_Add_bh := 0.0;
                ELSIF rtb_Add_no > 6553.5 THEN 
                    (* Switch: '<S614>/Switch1' incorporates:
                     *  Constant: '<S608>/Constant4' *)
                    rtb_Add_bh := 0.0;
                ELSE 
                    (* Switch: '<S614>/Switch1' *)
                    rtb_Add_bh := rtb_Add_no;
                END_IF;

                (* End of Switch: '<S614>/Switch' *)
            3: 
                rtb_Add_bh := 0.0;
            ELSE
                rtb_Add_bh := 0.0;
        END_CASE;

        (* End of MultiPortSwitch: '<S737>/Multiport Switch' *)
        

        (* MultiPortSwitch: '<S723>/Multiport Switch' incorporates:
         *  Constant: '<S723>/Constant'
         *  Delay: '<S723>/Delay' *)

        CASE TRUNC(rtb_BattSelect_f) OF
            1: 
                rtb_IP_boBMS_IMD_Active_BB1 := IP_boBatt1_IMD_active;
            2: 
                rtb_IP_boBMS_IMD_Active_BB1 := Delay_DSTATE_a[0];
            3: 
                rtb_IP_boBMS_IMD_Active_BB1 := FALSE;
            ELSE
                rtb_IP_boBMS_IMD_Active_BB1 := FALSE;
        END_CASE;

        (* End of MultiPortSwitch: '<S723>/Multiport Switch' *)
        

        (* MultiPortSwitch: '<S721>/Multiport Switch' incorporates:
         *  Constant: '<S721>/Constant'
         *  Delay: '<S721>/Delay' *)

        CASE TRUNC(rtb_BattSelect) OF
            1: 
                rtb_IP_boBMS_IMD_Active_BB2 := IP_boBatt2_IMD_active;
            2: 
                rtb_IP_boBMS_IMD_Active_BB2 := Delay_DSTATE_ov[0];
            3: 
                rtb_IP_boBMS_IMD_Active_BB2 := FALSE;
            ELSE
                rtb_IP_boBMS_IMD_Active_BB2 := FALSE;
        END_CASE;

        (* End of MultiPortSwitch: '<S721>/Multiport Switch' *)
        

        (* MultiPortSwitch: '<S722>/Multiport Switch' incorporates:
         *  Constant: '<S722>/Constant'
         *  Delay: '<S722>/Delay' *)

        CASE TRUNC(rtb_BattSelect_i) OF
            1: 
                rtb_IP_boBMS_IMD_Active_BB3 := IP_boBatt3_IMD_active;
            2: 
                rtb_IP_boBMS_IMD_Active_BB3 := Delay_DSTATE_c[0];
            3: 
                rtb_IP_boBMS_IMD_Active_BB3 := FALSE;
            ELSE
                rtb_IP_boBMS_IMD_Active_BB3 := FALSE;
        END_CASE;

        (* End of MultiPortSwitch: '<S722>/Multiport Switch' *)
        

        (* Sum: '<S223>/Add' incorporates:
         *  ArithShift: '<S222>/Shift Arithmetic'
         *  Constant: '<S211>/Constant'
         *  DataTypeConversion: '<S222>/Data Type Conversion'
         *  Product: '<S223>/Product'
         *  Sum: '<S222>/Add' *)
        rtb_Add_ci := DINT_TO_REAL(DWORD_TO_DINT(SHL(DINT_TO_DWORD(USINT_TO_DINT(C_Actia_Batt1_MyStatus[6])), 8)) + USINT_TO_DINT(C_Actia_Batt1_MyStatus[5])) * 0.02;
        (* Switch: '<S223>/Switch' incorporates:
         *  Constant: '<S211>/Constant3'
         *  Constant: '<S211>/SafeValue_NA '
         *  RelationalOperator: '<S223>/GreaterThan'
         *  Switch: '<S223>/Switch1' *)

        IF C_Actia_Batt1_MyStatus_Timeout THEN 
            rtb_Add_ci := 0.0;
        ELSIF rtb_Add_ci > 1310.7 THEN 
            (* Switch: '<S223>/Switch1' incorporates:
             *  Constant: '<S211>/SafeValue_Error' *)
            rtb_Add_ci := 0.0;
        END_IF;

        (* End of Switch: '<S223>/Switch' *)
        

        (* Sum: '<S284>/Add' incorporates:
         *  ArithShift: '<S283>/Shift Arithmetic'
         *  Constant: '<S272>/Constant'
         *  DataTypeConversion: '<S283>/Data Type Conversion'
         *  Product: '<S284>/Product'
         *  Sum: '<S283>/Add' *)
        rtb_UnitDelay := DINT_TO_REAL(DWORD_TO_DINT(SHL(DINT_TO_DWORD(USINT_TO_DINT(C_Actia_Batt2_MyStatus[6])), 8)) + USINT_TO_DINT(C_Actia_Batt2_MyStatus[5])) * 0.02;
        (* Switch: '<S284>/Switch' incorporates:
         *  Constant: '<S272>/Constant3'
         *  Constant: '<S272>/SafeValue_NA '
         *  RelationalOperator: '<S284>/GreaterThan'
         *  Switch: '<S284>/Switch1' *)

        IF C_Actia_Batt2_MyStatus_Timeout THEN 
            rtb_UnitDelay := 0.0;
        ELSIF rtb_UnitDelay > 1310.7 THEN 
            (* Switch: '<S284>/Switch1' incorporates:
             *  Constant: '<S272>/SafeValue_Error' *)
            rtb_UnitDelay := 0.0;
        END_IF;

        (* End of Switch: '<S284>/Switch' *)
        

        (* Sum: '<S345>/Add' incorporates:
         *  ArithShift: '<S344>/Shift Arithmetic'
         *  Constant: '<S333>/Constant'
         *  DataTypeConversion: '<S344>/Data Type Conversion'
         *  Product: '<S345>/Product'
         *  Sum: '<S344>/Add' *)
        rtb_Switch3 := DINT_TO_REAL(DWORD_TO_DINT(SHL(DINT_TO_DWORD(USINT_TO_DINT(C_Actia_Batt3_MyStatus[6])), 8)) + USINT_TO_DINT(C_Actia_Batt3_MyStatus[5])) * 0.02;
        (* Switch: '<S345>/Switch' incorporates:
         *  Constant: '<S333>/Constant3'
         *  Constant: '<S333>/SafeValue_NA '
         *  RelationalOperator: '<S345>/GreaterThan'
         *  Switch: '<S345>/Switch1' *)

        IF C_Actia_Batt3_MyStatus_Timeout THEN 
            rtb_Switch3 := 0.0;
        ELSIF rtb_Switch3 > 1310.7 THEN 
            (* Switch: '<S345>/Switch1' incorporates:
             *  Constant: '<S333>/SafeValue_Error' *)
            rtb_Switch3 := 0.0;
        END_IF;

        (* End of Switch: '<S345>/Switch' *)
        

        (* MultiPortSwitch: '<S772>/Multiport Switch' incorporates:
         *  Constant: '<S772>/Constant' *)

        CASE TRUNC(rtb_BattSelect_f) OF
            1: 
                rtb_IP_boBMS_Batt1_Availability := TRUNC(rtb_Uk1);
            2: 
                rtb_IP_boBMS_Batt1_Availability := BOOL_TO_DINT(rtb_Switch2_d);
            3: 
                rtb_IP_boBMS_Batt1_Availability := 0;
            ELSE
                rtb_IP_boBMS_Batt1_Availability := 0;
        END_CASE;

        (* End of MultiPortSwitch: '<S772>/Multiport Switch' *)
        

        (* MultiPortSwitch: '<S773>/Multiport Switch' incorporates:
         *  Constant: '<S773>/Constant' *)

        CASE TRUNC(rtb_BattSelect) OF
            1: 
                ;
                ;
            2: 
                rtb_UnitDelay5 := BOOL_TO_DINT(rtb_Switch1_fj);
            3: 
                rtb_UnitDelay5 := 0;
            ELSE
                rtb_UnitDelay5 := 0;
        END_CASE;

        (* End of MultiPortSwitch: '<S773>/Multiport Switch' *)
        

        (* MultiPortSwitch: '<S774>/Multiport Switch' incorporates:
         *  Constant: '<S774>/Constant' *)

        CASE TRUNC(rtb_BattSelect_i) OF
            1: 
                rtb_IP_boBMS_Batt3_Availability := TRUNC(rtb_Uk1);
            2: 
                rtb_IP_boBMS_Batt3_Availability := BOOL_TO_DINT(rtb_Switch_b);
            3: 
                rtb_IP_boBMS_Batt3_Availability := 0;
            ELSE
                rtb_IP_boBMS_Batt3_Availability := 0;
        END_CASE;

        (* End of MultiPortSwitch: '<S774>/Multiport Switch' *)
        

        (* Sum: '<S256>/Add' incorporates:
         *  ArithShift: '<S255>/Shift Arithmetic'
         *  Constant: '<S252>/Constant4'
         *  DataTypeConversion: '<S255>/Data Type Conversion'
         *  Product: '<S256>/Product'
         *  Sum: '<S255>/Add' *)
        rtb_Add_no := DINT_TO_REAL(DWORD_TO_DINT(SHL(DINT_TO_DWORD(USINT_TO_DINT(C_Actia_Batt1_ADS_1[4])), 8)) + USINT_TO_DINT(C_Actia_Batt1_ADS_1[3])) * 0.1;
        (* MultiPortSwitch: '<S741>/Multiport Switch' incorporates:
         *  Constant: '<S741>/Constant' *)

        CASE TRUNC(rtb_BattSelect_f) OF
            1: 
                (* Switch: '<S256>/Switch' incorporates:
                 *  Constant: '<S252>/Constant7'
                 *  Constant: '<S252>/Constant9'
                 *  RelationalOperator: '<S256>/GreaterThan'
                 *  Switch: '<S256>/Switch1' *)

                IF C_Actia_Batt1_ADS_1_Timeout THEN 
                    rtb_Add_no := 0.0;
                ELSIF rtb_Add_no > 125.0 THEN 
                    (* Switch: '<S256>/Switch1' incorporates:
                     *  Constant: '<S252>/Constant8' *)
                    rtb_Add_no := 0.0;
                END_IF;

                (* End of Switch: '<S256>/Switch' *)
            2: 
                (* Switch: '<S440>/Switch' incorporates:
                 *  Constant: '<S433>/Constant4' *)

                IF C_LB_Batt1_CellTemperature_Timeout THEN 
                    rtb_Add_no := 0.0;
                ELSE 
                    (* Switch: '<S440>/Switch1' incorporates:
                     *  DataTypeConversion: '<S433>/Data Type Conversion' *)
                    rtb_Add_no := SINT_TO_REAL(USINT_TO_SINT(C_LB_Batt1_CellTemperature_Msg[1]));
                END_IF;

                (* End of Switch: '<S440>/Switch' *)
            3: 
                rtb_Add_no := 0.0;
            ELSE
                rtb_Add_no := 0.0;
        END_CASE;

        (* End of MultiPortSwitch: '<S741>/Multiport Switch' *)
        

        (* Sum: '<S258>/Add' incorporates:
         *  ArithShift: '<S257>/Shift Arithmetic'
         *  Constant: '<S253>/Constant4'
         *  DataTypeConversion: '<S257>/Data Type Conversion'
         *  Product: '<S258>/Product'
         *  Sum: '<S257>/Add' *)
        rtb_Add_a5 := DINT_TO_REAL(DWORD_TO_DINT(SHL(DINT_TO_DWORD(USINT_TO_DINT(C_Actia_Batt1_ADS_1[6])), 8)) + USINT_TO_DINT(C_Actia_Batt1_ADS_1[5])) * 0.1;
        (* MultiPortSwitch: '<S739>/Multiport Switch' incorporates:
         *  Constant: '<S739>/Constant' *)

        CASE TRUNC(rtb_BattSelect_f) OF
            1: 
                (* Switch: '<S258>/Switch' incorporates:
                 *  Constant: '<S253>/Constant7'
                 *  Constant: '<S253>/Constant9'
                 *  RelationalOperator: '<S258>/GreaterThan'
                 *  Switch: '<S258>/Switch1' *)

                IF C_Actia_Batt1_ADS_1_Timeout THEN 
                    rtb_Add_a5 := 0.0;
                ELSIF rtb_Add_a5 > 125.0 THEN 
                    (* Switch: '<S258>/Switch1' incorporates:
                     *  Constant: '<S253>/Constant8' *)
                    rtb_Add_a5 := 0.0;
                END_IF;

                (* End of Switch: '<S258>/Switch' *)
            2: 
                (* Switch: '<S441>/Switch' incorporates:
                 *  Constant: '<S434>/Constant4' *)

                IF C_LB_Batt1_CellTemperature_Timeout THEN 
                    rtb_Add_a5 := 0.0;
                ELSE 
                    (* Switch: '<S441>/Switch1' incorporates:
                     *  DataTypeConversion: '<S434>/Data Type Conversion' *)
                    rtb_Add_a5 := SINT_TO_REAL(USINT_TO_SINT(C_LB_Batt1_CellTemperature_Msg[2]));
                END_IF;

                (* End of Switch: '<S441>/Switch' *)
            3: 
                rtb_Add_a5 := 0.0;
            ELSE
                rtb_Add_a5 := 0.0;
        END_CASE;

        (* End of MultiPortSwitch: '<S739>/Multiport Switch' *)
        

        (* Sum: '<S320>/Add' incorporates:
         *  ArithShift: '<S319>/Shift Arithmetic'
         *  Constant: '<S315>/Constant4'
         *  DataTypeConversion: '<S319>/Data Type Conversion'
         *  Product: '<S320>/Product'
         *  Sum: '<S319>/Add' *)
        rtb_Add_g4 := DINT_TO_REAL(DWORD_TO_DINT(SHL(DINT_TO_DWORD(USINT_TO_DINT(C_Actia_Batt2_ADS_1[4])), 8)) + USINT_TO_DINT(C_Actia_Batt2_ADS_1[3])) * 0.1;
        (* MultiPortSwitch: '<S740>/Multiport Switch' incorporates:
         *  Constant: '<S740>/Constant' *)

        CASE TRUNC(rtb_BattSelect) OF
            1: 
                (* Switch: '<S320>/Switch' incorporates:
                 *  Constant: '<S315>/Constant7'
                 *  Constant: '<S315>/Constant9'
                 *  RelationalOperator: '<S320>/GreaterThan'
                 *  Switch: '<S320>/Switch1' *)

                IF C_Actia_Batt2_ADS_1_Timeout THEN 
                    rtb_Add_g4 := 0.0;
                ELSIF rtb_Add_g4 > 125.0 THEN 
                    (* Switch: '<S320>/Switch1' incorporates:
                     *  Constant: '<S315>/Constant8' *)
                    rtb_Add_g4 := 0.0;
                END_IF;

                (* End of Switch: '<S320>/Switch' *)
            2: 
                (* Switch: '<S520>/Switch' incorporates:
                 *  Constant: '<S513>/Constant4' *)

                IF C_LB_Batt2_CellTemperature_Timeout THEN 
                    rtb_Add_g4 := 0.0;
                ELSE 
                    (* Switch: '<S520>/Switch1' incorporates:
                     *  DataTypeConversion: '<S513>/Data Type Conversion' *)
                    rtb_Add_g4 := SINT_TO_REAL(USINT_TO_SINT(C_LB_Batt2_CellTemperature_Msg[1]));
                END_IF;

                (* End of Switch: '<S520>/Switch' *)
            3: 
                rtb_Add_g4 := 0.0;
            ELSE
                rtb_Add_g4 := 0.0;
        END_CASE;

        (* End of MultiPortSwitch: '<S740>/Multiport Switch' *)
        

        (* Sum: '<S317>/Add' incorporates:
         *  ArithShift: '<S316>/Shift Arithmetic'
         *  Constant: '<S313>/Constant4'
         *  DataTypeConversion: '<S316>/Data Type Conversion'
         *  Product: '<S317>/Product'
         *  Sum: '<S316>/Add' *)
        rtb_Add_i5o := DINT_TO_REAL(DWORD_TO_DINT(SHL(DINT_TO_DWORD(USINT_TO_DINT(C_Actia_Batt2_ADS_1[6])), 8)) + USINT_TO_DINT(C_Actia_Batt2_ADS_1[5])) * 0.1;
        (* MultiPortSwitch: '<S742>/Multiport Switch' incorporates:
         *  Constant: '<S742>/Constant' *)

        CASE TRUNC(rtb_BattSelect) OF
            1: 
                (* Switch: '<S317>/Switch' incorporates:
                 *  Constant: '<S313>/Constant7'
                 *  Constant: '<S313>/Constant9'
                 *  RelationalOperator: '<S317>/GreaterThan'
                 *  Switch: '<S317>/Switch1' *)

                IF C_Actia_Batt2_ADS_1_Timeout THEN 
                    rtb_Add_i5o := 0.0;
                ELSIF rtb_Add_i5o > 125.0 THEN 
                    (* Switch: '<S317>/Switch1' incorporates:
                     *  Constant: '<S313>/Constant8' *)
                    rtb_Add_i5o := 0.0;
                END_IF;

                (* End of Switch: '<S317>/Switch' *)
            2: 
                (* Switch: '<S521>/Switch' incorporates:
                 *  Constant: '<S514>/Constant4' *)

                IF C_LB_Batt2_CellTemperature_Timeout THEN 
                    rtb_Add_i5o := 0.0;
                ELSE 
                    (* Switch: '<S521>/Switch1' incorporates:
                     *  DataTypeConversion: '<S514>/Data Type Conversion' *)
                    rtb_Add_i5o := SINT_TO_REAL(USINT_TO_SINT(C_LB_Batt2_CellTemperature_Msg[2]));
                END_IF;

                (* End of Switch: '<S521>/Switch' *)
            3: 
                rtb_Add_i5o := 0.0;
            ELSE
                rtb_Add_i5o := 0.0;
        END_CASE;

        (* End of MultiPortSwitch: '<S742>/Multiport Switch' *)
        

        (* Sum: '<S378>/Add' incorporates:
         *  ArithShift: '<S377>/Shift Arithmetic'
         *  Constant: '<S374>/Constant4'
         *  DataTypeConversion: '<S377>/Data Type Conversion'
         *  Product: '<S378>/Product'
         *  Sum: '<S377>/Add' *)
        rtb_Add_pi := DINT_TO_REAL(DWORD_TO_DINT(SHL(DINT_TO_DWORD(USINT_TO_DINT(C_Actia_Batt3_ADS_1[4])), 8)) + USINT_TO_DINT(C_Actia_Batt3_ADS_1[3])) * 0.1;
        (* MultiPortSwitch: '<S743>/Multiport Switch' incorporates:
         *  Constant: '<S743>/Constant' *)

        CASE TRUNC(rtb_BattSelect_i) OF
            1: 
                (* Switch: '<S378>/Switch' incorporates:
                 *  Constant: '<S374>/Constant7'
                 *  Constant: '<S374>/Constant9'
                 *  RelationalOperator: '<S378>/GreaterThan'
                 *  Switch: '<S378>/Switch1' *)

                IF C_Actia_Batt3_ADS_1_Timeout THEN 
                    rtb_Add_pi := 0.0;
                ELSIF rtb_Add_pi > 125.0 THEN 
                    (* Switch: '<S378>/Switch1' incorporates:
                     *  Constant: '<S374>/Constant8' *)
                    rtb_Add_pi := 0.0;
                END_IF;

                (* End of Switch: '<S378>/Switch' *)
            2: 
                (* Switch: '<S600>/Switch' incorporates:
                 *  Constant: '<S593>/Constant4' *)

                IF C_LB_Batt3_CellTemperature_Timeout THEN 
                    rtb_Add_pi := 0.0;
                ELSE 
                    (* Switch: '<S600>/Switch1' incorporates:
                     *  DataTypeConversion: '<S593>/Data Type Conversion' *)
                    rtb_Add_pi := SINT_TO_REAL(USINT_TO_SINT(C_LB_Batt3_CellTemperature_Msg[1]));
                END_IF;

                (* End of Switch: '<S600>/Switch' *)
            3: 
                rtb_Add_pi := 0.0;
            ELSE
                rtb_Add_pi := 0.0;
        END_CASE;

        (* End of MultiPortSwitch: '<S743>/Multiport Switch' *)
        

        (* Sum: '<S380>/Add' incorporates:
         *  ArithShift: '<S379>/Shift Arithmetic'
         *  Constant: '<S375>/Constant4'
         *  DataTypeConversion: '<S379>/Data Type Conversion'
         *  Product: '<S380>/Product'
         *  Sum: '<S379>/Add' *)
        rtb_Add_eo := DINT_TO_REAL(DWORD_TO_DINT(SHL(DINT_TO_DWORD(USINT_TO_DINT(C_Actia_Batt3_ADS_1[6])), 8)) + USINT_TO_DINT(C_Actia_Batt3_ADS_1[5])) * 0.1;
        (* MultiPortSwitch: '<S744>/Multiport Switch' incorporates:
         *  Constant: '<S744>/Constant' *)

        CASE TRUNC(rtb_BattSelect_i) OF
            1: 
                (* Switch: '<S380>/Switch' incorporates:
                 *  Constant: '<S375>/Constant7'
                 *  Constant: '<S375>/Constant9'
                 *  RelationalOperator: '<S380>/GreaterThan'
                 *  Switch: '<S380>/Switch1' *)

                IF C_Actia_Batt3_ADS_1_Timeout THEN 
                    rtb_Add_eo := 0.0;
                ELSIF rtb_Add_eo > 125.0 THEN 
                    (* Switch: '<S380>/Switch1' incorporates:
                     *  Constant: '<S375>/Constant8' *)
                    rtb_Add_eo := 0.0;
                END_IF;

                (* End of Switch: '<S380>/Switch' *)
            2: 
                (* Switch: '<S601>/Switch' incorporates:
                 *  Constant: '<S594>/Constant4' *)

                IF C_LB_Batt3_CellTemperature_Timeout THEN 
                    rtb_Add_eo := 0.0;
                ELSE 
                    (* Switch: '<S601>/Switch1' incorporates:
                     *  DataTypeConversion: '<S594>/Data Type Conversion' *)
                    rtb_Add_eo := SINT_TO_REAL(USINT_TO_SINT(C_LB_Batt3_CellTemperature_Msg[2]));
                END_IF;

                (* End of Switch: '<S601>/Switch' *)
            3: 
                rtb_Add_eo := 0.0;
            ELSE
                rtb_Add_eo := 0.0;
        END_CASE;

        (* End of MultiPortSwitch: '<S744>/Multiport Switch' *)
        

        (* Outputs for Atomic SubSystem: '<S676>/BatteryPackSignals' *)
        (* SignalConversion: '<S682>/BusConversion_InsertedFor_IT_BatterySignal_Databus_at_inport_0' *)
        rtb_IT_boBMS_Error_BB1 := IP_boBatt1_ERROR_activ;
        (* SignalConversion: '<S682>/BusConversion_InsertedFor_IT_BatterySignal_Databus_at_inport_0' *)
        rtb_IT_boBMS_Error_BB2 := IP_boBatt2_ERROR_activ;
        (* SignalConversion: '<S682>/BusConversion_InsertedFor_IT_BatterySignal_Databus_at_inport_0' *)
        rtb_IT_boBMS_Error_BB3 := IP_boBatt3_ERROR_activ;
        (* SignalConversion: '<S682>/BusConversion_InsertedFor_IT_BatterySignal_Databus_at_inport_0' *)
        rtb_IT_boBMS_Warning_BB1 := IP_boBatt1_WARNING_activ;
        (* SignalConversion: '<S682>/BusConversion_InsertedFor_IT_BatterySignal_Databus_at_inport_0' *)
        rtb_IT_boBMS_Warning_BB2 := IP_boBatt2_WARNING_activ;
        (* SignalConversion: '<S682>/BusConversion_InsertedFor_IT_BatterySignal_Databus_at_inport_0' *)
        rtb_IT_boBMS_Warning_BB3 := IP_boBatt3_WARNING_activ;
        (* Gain: '<S682>/Gain1' *)
        rtb_Add_c0 := 0.001 * rtb_Add_c0;
        (* Gain: '<S682>/Gain2' *)
        rtb_Add_egs := 0.001 * rtb_Add_egs;
        (* Gain: '<S682>/Gain3' *)
        rtb_IT_sBMS_InternalResistance_BB1_ohms := 0.001 * rtb_Switch_a;
        (* Logic: '<S682>/OR' *)
        rtb_IT_boBMS_HV_ON_BB := (rtb_IP_boBMS_HV_REL_ON_BB1 OR rtb_IP_boBMS_HV_REL_ON_BB2) OR rtb_IP_boBMS_HV_REL_ON_BB3;
        (* Sum: '<S701>/Add' incorporates:
         *  Logic: '<S701>/AND'
         *  Logic: '<S701>/AND1'
         *  Logic: '<S701>/AND2'
         *  Logic: '<S701>/NOT'
         *  Logic: '<S701>/NOT1'
         *  Logic: '<S701>/NOT2'
         *  SignalConversion: '<S698>/Signal Copy'
         *  SignalConversion: '<S699>/Signal Copy'
         *  SignalConversion: '<S700>/Signal Copy' *)
        rtb_ExtractDesiredBits_b13 := UDINT_TO_USINT((BOOL_TO_UDINT((rtb_IP_boBMS_Batt1_Availability <> 0) AND ( NOT rtb_IP_boBMS_SDError_BB1)) + BOOL_TO_UDINT((rtb_UnitDelay5 <> 0) AND ( NOT rtb_IP_boBMS_SDError_BB2))) + BOOL_TO_UDINT((rtb_IP_boBMS_Batt3_Availability <> 0) AND ( NOT rtb_IP_boBMS_SDError_BB3)));
        (* Logic: '<S702>/NOT' *)
        i0_IMDOK_Input_Delay(ssMethodType := SS_OUTPUT, In :=  NOT rtb_S_in);
        rtb_out_l := i0_IMDOK_Input_Delay.out;
        (* Logic: '<S702>/AND' *)
        rtb_AND_l2 := rtb_out_l AND (rtb_IP_boBMS_Batt1_Availability <> 0);
        (* Logic: '<S703>/NOT' *)
        i1_IMDOK_Input_Delay(ssMethodType := SS_OUTPUT, In :=  NOT rtb_IP_boBatt1_Actia_Availability);
        rtb_out_l := i1_IMDOK_Input_Delay.out;
        (* Logic: '<S703>/AND' *)
        rtb_AND_ni := rtb_out_l AND (rtb_UnitDelay5 <> 0);
        (* Logic: '<S704>/NOT' *)
        i2_IMDOK_Input_Delay(ssMethodType := SS_OUTPUT, In :=  NOT rtb_Delay_dl);
        rtb_out_l := i2_IMDOK_Input_Delay.out;
        (* Logic: '<S704>/AND' *)
        rtb_AND_ma := rtb_out_l AND (rtb_IP_boBMS_Batt3_Availability <> 0);
        (* SignalConversion: '<S698>/Signal Copy' incorporates:
         *  SignalConversion: '<S699>/Signal Copy'
         *  SignalConversion: '<S700>/Signal Copy' *)
        i0_VoltageDetermination(IP_sBMS_VtgInt_BB1 := rtb_Min, IP_sBMS_VtgInt_BB2 := rtb_Add_an, IP_sBMS_VtgInt_BB3 := rtb_Add_e, IP_boBMS_SDError_BB1 := rtb_IP_boBMS_SDError_BB1, IP_boBMS_SDError_BB2 := rtb_IP_boBMS_SDError_BB2, IP_boBMS_SDError_BB3 := rtb_IP_boBMS_SDError_BB3, IP_boBMS_Batt1_Availability := DINT_TO_LREAL(rtb_IP_boBMS_Batt1_Availability), IP_boBMS_Batt2_Availability := DINT_TO_LREAL(rtb_UnitDelay5), IP_boBMS_Batt3_Availability := DINT_TO_LREAL(rtb_IP_boBMS_Batt3_Availability));
        rtb_Switch_a := i0_VoltageDetermination.IT_u8BMS_BB_No_MaxVoltage;
        rtb_Switch2_k := i0_VoltageDetermination.IT_u8BMS_BB_No_MinVoltage;
        (* End of Outputs for SubSystem: '<S676>/BatteryPackSignals' *)
        

        (* Switch: '<S36>/Switch' incorporates:
         *  Constant: '<S36>/VoltageSensorAvailableBB1'
         *  Product: '<S36>/Product2'
         *  SignalConversion: '<S682>/BusConversion_InsertedFor_IT_BatterySignal_Databus_at_inport_0'
         *  Sum: '<S36>/Add' *)

        IF  NOT VoltageSensorAvailableBB1 THEN 
            (* Outputs for Atomic SubSystem: '<S676>/BatteryPackSignals' *)
            (* Switch: '<S36>/Switch3' incorporates:
             *  Constant: '<S36>/Constant'
             *  SignalConversion: '<S682>/BusConversion_InsertedFor_IT_BatterySignal_Databus_at_inport_0' *)

            IF rtb_IP_boBMS_HV_REL_ON_BB1 THEN 
                rtb_Add_ci := rtb_Add_ki5;
            ELSE 
                rtb_Add_ci := 0.0;
            END_IF;

            (* End of Switch: '<S36>/Switch3' *)
            rtb_Add_ci := rtb_Min - (rtb_IT_sBMS_InternalResistance_BB1_ohms * rtb_Add_ci);
            (* End of Outputs for SubSystem: '<S676>/BatteryPackSignals' *)
        END_IF;

        (* End of Switch: '<S36>/Switch' *)
        

        (* Switch: '<S36>/Switch1' incorporates:
         *  Constant: '<S36>/VoltageSensorAvailableBB2'
         *  Product: '<S36>/Product3'
         *  SignalConversion: '<S682>/BusConversion_InsertedFor_IT_BatterySignal_Databus_at_inport_0'
         *  Sum: '<S36>/Add1' *)

        IF  NOT VoltageSensorAvailableBB2 THEN 
            (* Outputs for Atomic SubSystem: '<S676>/BatteryPackSignals' *)
            (* Switch: '<S36>/Switch4' incorporates:
             *  Constant: '<S36>/Constant1'
             *  SignalConversion: '<S682>/BusConversion_InsertedFor_IT_BatterySignal_Databus_at_inport_0' *)

            IF rtb_IP_boBMS_HV_REL_ON_BB2 THEN 
                rtb_UnitDelay := rtb_Add_ir;
            ELSE 
                rtb_UnitDelay := 0.0;
            END_IF;

            (* End of Switch: '<S36>/Switch4' *)
            rtb_UnitDelay := rtb_Add_an - (rtb_Add_c0 * rtb_UnitDelay);
            (* End of Outputs for SubSystem: '<S676>/BatteryPackSignals' *)
        END_IF;

        (* End of Switch: '<S36>/Switch1' *)
        

        (* Switch: '<S36>/Switch2' incorporates:
         *  Constant: '<S36>/VoltageSensorAvailableBB3'
         *  Product: '<S36>/Product1'
         *  SignalConversion: '<S682>/BusConversion_InsertedFor_IT_BatterySignal_Databus_at_inport_0'
         *  Sum: '<S36>/Add2' *)

        IF  NOT VoltageSensorAvailableBB3 THEN 
            (* Outputs for Atomic SubSystem: '<S676>/BatteryPackSignals' *)
            (* Switch: '<S36>/Switch5' incorporates:
             *  Constant: '<S36>/Constant2'
             *  SignalConversion: '<S682>/BusConversion_InsertedFor_IT_BatterySignal_Databus_at_inport_0' *)

            IF rtb_IP_boBMS_HV_REL_ON_BB3 THEN 
                rtb_Switch3 := rtb_Add_m;
            ELSE 
                rtb_Switch3 := 0.0;
            END_IF;

            (* End of Switch: '<S36>/Switch5' *)
            rtb_Switch3 := rtb_Add_e - (rtb_Add_egs * rtb_Switch3);
            (* End of Outputs for SubSystem: '<S676>/BatteryPackSignals' *)
        END_IF;

        (* End of Switch: '<S36>/Switch2' *)
        

        (* Outputs for Atomic SubSystem: '<S676>/BatteryPackSignals' *)
        (* SignalConversion: '<S682>/BusConversion_InsertedFor_IT_BatterySignal_Databus_at_inport_0' *)
        i0_SafeToCloseHV(FL_sVtgExt_BB1 := rtb_Add_ci, FL_sVtgExt_BB2 := rtb_UnitDelay, FL_sVtgExt_BB3 := rtb_Switch3, VtgInt_BB1 := rtb_Min, VtgInt_BB2 := rtb_Add_an, VtgInt_BB3 := rtb_Add_e, IMD_Active_BB1 := rtb_IP_boBMS_IMD_Active_BB1, IMD_Active_BB2 := rtb_IP_boBMS_IMD_Active_BB2, IMD_Active_BB3 := rtb_IP_boBMS_IMD_Active_BB3, InternalResistance_BB1 := rtb_IT_sBMS_InternalResistance_BB1_ohms, InternalResistance_BB2 := rtb_Add_c0, InternalResistance_BB3 := rtb_Add_egs, HV_REL_ON_BB1 := rtb_IP_boBMS_HV_REL_ON_BB1, HV_REL_ON_BB2 := rtb_IP_boBMS_HV_REL_ON_BB2, HV_REL_ON_BB3 := rtb_IP_boBMS_HV_REL_ON_BB3);
        rtb_Delay_j := i0_SafeToCloseHV.FL_boSafeToCloseHV_BB1;
        rtb_FL_boSS_HVIL_NOK := i0_SafeToCloseHV.FL_boSafeToCloseHV_BB2;
        rtb_FL_boHVC_AllCellBalanced := i0_SafeToCloseHV.FL_boSafeToCloseHV_BB3;
        rtb_Abs := i0_SafeToCloseHV.FL_sCalculated_Vtg_Diff_BB1;
        rtb_Abs1 := i0_SafeToCloseHV.FL_sCalculated_Vtg_Diff_BB2;
        rtb_Abs2 := i0_SafeToCloseHV.FL_sCalculated_Vtg_Diff_BB3;
        rtb_Divide_i := i0_SafeToCloseHV.FL_sCalculated_InrushCurrent_BB1;
        rtb_Divide1_p := i0_SafeToCloseHV.FL_sCalculated_InrushCurrent_BB2;
        rtb_Divide2 := i0_SafeToCloseHV.FL_sCalculated_InrushCurrent_BB3;
        (* End of Outputs for SubSystem: '<S676>/BatteryPackSignals' *)
        

        (* UnitDelay: '<S35>/Unit Delay1' *)
        rtb_Uk1 := UnitDelay1_DSTATE_f;
        (* RelationalOperator: '<S44>/Compare' incorporates:
         *  Constant: '<S44>/Constant' *)
        rtb_Switch_b := rtb_Uk1 = 1.0;
        (* Logic: '<S35>/OR' incorporates:
         *  Constant: '<S43>/Constant'
         *  RelationalOperator: '<S43>/Compare' *)
        rtb_out_l := rtb_Switch_b OR (rtb_Uk1 = 3.0);
        (* UnitDelay: '<S35>/Unit Delay' *)
        rtb_Uk1 := UnitDelay_DSTATE_o;
        (* RelationalOperator: '<S46>/Compare' incorporates:
         *  Constant: '<S46>/Constant' *)
        rtb_Switch1_fj := rtb_Uk1 = 1.0;
        (* Outputs for Atomic SubSystem: '<S676>/BatteryPackSignals' *)
        (* SignalConversion: '<S8>/TmpSignal ConversionAtREQ_HV_ON_BattInport3' incorporates:
         *  Constant: '<S45>/Constant'
         *  Logic: '<S35>/AND'
         *  Logic: '<S35>/NOT'
         *  Logic: '<S35>/OR1'
         *  Logic: '<S35>/OR2'
         *  Logic: '<S8>/OR'
         *  RelationalOperator: '<S45>/Compare'
         *  RelationalOperator: '<S47>/Compare'
         *  SignalConversion: '<S682>/BusConversion_InsertedFor_IT_BatterySignal_Databus_at_inport_0'
         *  SignalConversion: '<S698>/Signal Copy'
         *  SignalConversion: '<S699>/Signal Copy'
         *  SignalConversion: '<S700>/Signal Copy'
         *  SignalConversion: '<S8>/TmpSignal ConversionAtREQ_HV_ON_BattInport4'
         *  UnitDelay: '<S35>/Unit Delay2'
         *  UnitDelay: '<S8>/Unit Delay1'
         *  UnitDelay: '<S8>/Unit Delay2'
         *  UnitDelay: '<S8>/Unit Delay3'
         *  UnitDelay: '<S8>/Unit Delay4'
         *  UnitDelay: '<S8>/Unit Delay5'
         *  UnitDelay: '<S8>/Unit Delay6'
         *  UnitDelay: '<S8>/Unit Delay7'
         *  UnitDelay: '<S8>/Unit Delay9' *)
        i0_REQ_HV_ON_Batt(ssMethodType := SS_OUTPUT, IsolationMeasurementRequest := rtb_IT_boUDC_EV_IsolationMeasurementRequest, IP_boChargeStop_Pressed := rtb_IT_boChargeStop_Button, SafeToSD_BB1 := rtb_FL_boCMSleep, SafeToSD_BB2 := rtb_FL_boCMSleep, SafeToSD_BB3 := rtb_FL_boCMSleep, KL15_CM_disable := rtb_FL_boKL15_Disable, SDError_BB1 := rtb_IP_boBMS_SDError_BB1, SDError_BB2 := rtb_IP_boBMS_SDError_BB2, SDError_BB3 := rtb_IP_boBMS_SDError_BB3, InsulationReadyOK_B1 := rtb_S_in, InsulationReadyOK_B2 := rtb_IP_boBatt1_Actia_Availability, InsulationReadyOK_B3 := rtb_Delay_dl, IMD_Active_BB1 := rtb_IP_boBMS_IMD_Active_BB1, IMD_Active_BB2 := rtb_IP_boBMS_IMD_Active_BB2, IMD_Active_BB3 := rtb_IP_boBMS_IMD_Active_BB3, Software_Reset_KL15_BB3 := UnitDelay5_DSTATE, Software_Reset_KL15_BB2 := UnitDelay4_DSTATE, Software_Reset_KL15_BB1 := UnitDelay3_DSTATE, FL_boSafeToCloseHV_BB1 := rtb_Delay_j, FL_boSafeToCloseHV_BB2 := rtb_FL_boSS_HVIL_NOK, FL_boSafeToCloseHV_BB3 := rtb_FL_boHVC_AllCellBalanced, FL_boST_REQ_HV_Open_BB1 := UnitDelay2_DSTATE_d, FL_boST_REQ_HV_Open_BB2 := UnitDelay6_DSTATE_b, FL_boST_REQ_HV_Open_BB3 := UnitDelay7_DSTATE_j, FL_boSystem_SD := UnitDelay9_DSTATE OR UnitDelay1_DSTATE_fl, HV_Minus_Sense_BB1 := rtb_IP_boBMS_HV_Minus_Sense_BB1, HV_Plus_Sense_BB1 := rtb_IP_boBMS_HV_Plus_Sense_BB1, HV_Minus_Sense_BB2 := rtb_IP_boBMS_HV_Minus_Sense_BB2, HV_Plus_Sense_BB2 := rtb_IP_boBMS_HV_Plus_Sense_BB2, HV_Minus_Sense_BB3 := rtb_IP_boBMS_HV_Minus_Sense_BB3, HV_Plus_Sense_BB3 := rtb_IP_boBMS_HV_Plus_Sense_BB3, HV_REL_ON_BB2 := rtb_IP_boBMS_HV_REL_ON_BB1, HV_REL_ON_BB1 := rtb_IP_boBMS_HV_REL_ON_BB2, HV_REL_ON_BB3 := rtb_IP_boBMS_HV_REL_ON_BB3, FL_boMainHV_SD_OK := (rtb_out_l AND (rtb_Switch1_fj OR (rtb_Uk1 = 3.0))) AND ( NOT UnitDelay2_DSTATE_g), FL_boMainHV_PlusMinus_Status := ( NOT rtb_Switch_b) OR ( NOT rtb_Switch1_fj));
        ContactorState_i := i0_REQ_HV_ON_Batt.FL_u8ContactorState_BB1;
        ContactorState_f := i0_REQ_HV_ON_Batt.FL_u8ContactorState_BB2;
        ContactorState := i0_REQ_HV_ON_Batt.FL_u8ContactorState_BB3;
        REQ_HV_ON_a := i0_REQ_HV_ON_Batt.FL_boREQ_HV_ON_BB1;
        REQ_HV_ON_d := i0_REQ_HV_ON_Batt.FL_boREQ_HV_ON_BB2;
        REQ_HV_ON := i0_REQ_HV_ON_Batt.FL_boREQ_HV_ON_BB3;
        rtb_Contactor_FB_State_h := i0_REQ_HV_ON_Batt.FL_u8Contactor_FB_State_BB1;
        rtb_Contactor_FB_State_g := i0_REQ_HV_ON_Batt.FL_u8Contactor_FB_State_BB2;
        rtb_Contactor_FB_State := i0_REQ_HV_ON_Batt.FL_u8Contactor_FB_State_BB3;
        (* Logic: '<S13>/AND' incorporates:
         *  SignalConversion: '<S682>/BusConversion_InsertedFor_IT_BatterySignal_Databus_at_inport_0' *)
        rtb_Delay_j := (REQ_HV_ON_a <> 0.0) AND rtb_IP_boBMS_HV_REL_ON_BB1;
        (* Logic: '<S13>/AND1' incorporates:
         *  SignalConversion: '<S682>/BusConversion_InsertedFor_IT_BatterySignal_Databus_at_inport_0' *)
        rtb_FL_boSS_HVIL_NOK := (REQ_HV_ON_d <> 0.0) AND rtb_IP_boBMS_HV_REL_ON_BB2;
        (* Logic: '<S13>/AND2' incorporates:
         *  SignalConversion: '<S682>/BusConversion_InsertedFor_IT_BatterySignal_Databus_at_inport_0' *)
        rtb_out_l := (REQ_HV_ON <> 0.0) AND rtb_IP_boBMS_HV_REL_ON_BB3;
        (* End of Outputs for SubSystem: '<S676>/BatteryPackSignals' *)
        

        (* UnitDelay: '<S13>/Unit Delay3' *)
        rtb_Uk1 := UnitDelay3_DSTATE_p;
        (* Logic: '<S13>/AND3' incorporates:
         *  SignalConversion: '<S678>/Signal Copy4' *)
        DO_REQ_DC_ON_PLUS := (rtb_Uk1 <> 0.0) AND IP_boEVDisconnectingDevice;
        (* UnitDelay: '<S13>/Unit Delay2' *)
        rtb_UnitDelay2 := UnitDelay2_DSTATE_a;
        (* Chart: '<S13>/Chart_REQ_MAIN_Precharge' incorporates:
         *  UnitDelay: '<S13>/Unit Delay6' *)
        (* Gateway: ChiefMaster/Flow Logic/BDU Control/BDUSystem/Chart_REQ_MAIN_Precharge *)
        (* During: ChiefMaster/Flow Logic/BDU Control/BDUSystem/Chart_REQ_MAIN_Precharge *)

        IF is_active_c19_ChiefMaster = 0 THEN 
            (* Entry: ChiefMaster/Flow Logic/BDU Control/BDUSystem/Chart_REQ_MAIN_Precharge *)
            is_active_c19_ChiefMaster := 1;
            (* Entry Internal: ChiefMaster/Flow Logic/BDU Control/BDUSystem/Chart_REQ_MAIN_Precharge *)
            (* Transition: '<S17>:4' *)
            is_c19_ChiefMaster := ChiefMaster_IN_Default_e2;
            (* Entry 'Default': '<S17>:3' *)
            (* '<S17>:3:2' REQ_MainHV_ON_Precharge = false *)
            DO_REQ_MainHV_ON_Precharge := FALSE;
        ELSE 

            CASE is_c19_ChiefMaster OF
                ChiefMaster_IN_Default_e2: 
                    (* During 'Default': '<S17>:3' *)
                    (* '<S17>:7:1' sf_internal_predicateOutput = MainHV_Minus_Status == 2 &&... *)
                    (* '<S17>:7:2' KL15_CM_disable == false; *)

                    IF (rtb_UnitDelay2 = 2.0) AND ( NOT rtb_FL_boKL15_Disable) THEN 
                        (* Transition: '<S17>:7' *)
                        is_c19_ChiefMaster := ChiefMaster_IN_PrechargeEnable;
                        (* Entry 'PrechargeEnable': '<S17>:6' *)
                        (* '<S17>:6:2' REQ_MainHV_ON_Precharge = true *)
                        DO_REQ_MainHV_ON_Precharge := TRUE;
                    ELSE 
                        (* '<S17>:3:2' REQ_MainHV_ON_Precharge = false *)
                        DO_REQ_MainHV_ON_Precharge := FALSE;
                    END_IF;

                ChiefMaster_IN_PrechargeDisable: 
                    (* During 'PrechargeDisable': '<S17>:10' *)
                    (* '<S17>:12:1' sf_internal_predicateOutput = KL15_CM_disable == true ||... *)
                    (* '<S17>:12:2' (MainHV_Minus_Status == 1 || MainHV_Minus_Status == 3); *)

                    IF (rtb_FL_boKL15_Disable OR (rtb_UnitDelay2 = 1.0)) OR (rtb_UnitDelay2 = 3.0) THEN 
                        (* Transition: '<S17>:12' *)
                        is_c19_ChiefMaster := ChiefMaster_IN_Default_e2;
                        (* Entry 'Default': '<S17>:3' *)
                        (* '<S17>:3:2' REQ_MainHV_ON_Precharge = false *)
                        DO_REQ_MainHV_ON_Precharge := FALSE;
                    ELSE 
                        (* '<S17>:10:2' REQ_MainHV_ON_Precharge = false *)
                        DO_REQ_MainHV_ON_Precharge := FALSE;
                    END_IF;

                ELSE
                    (* During 'PrechargeEnable': '<S17>:6' *)
                    (* '<S17>:11:1' sf_internal_predicateOutput = System_SD == true ||... *)
                    (* '<S17>:11:2' (MainHV_Plus_Status == 2 || MainHV_Plus_Status == 3) ||... *)
                    (* '<S17>:11:3' (MainHV_Minus_Status == 1 || MainHV_Minus_Status == 3); *)

                    IF (((UnitDelay6_DSTATE_h OR (rtb_Uk1 = 2.0)) OR (rtb_Uk1 = 3.0)) OR (rtb_UnitDelay2 = 1.0)) OR (rtb_UnitDelay2 = 3.0) THEN 
                        (* Transition: '<S17>:11' *)
                        is_c19_ChiefMaster := ChiefMaster_IN_PrechargeDisable;
                        (* Entry 'PrechargeDisable': '<S17>:10' *)
                        (* '<S17>:10:2' REQ_MainHV_ON_Precharge = false *)
                        DO_REQ_MainHV_ON_Precharge := FALSE;
                    ELSE 
                        (* '<S17>:6:2' REQ_MainHV_ON_Precharge = true *)
                        DO_REQ_MainHV_ON_Precharge := TRUE;
                    END_IF;

            END_CASE;

        END_IF;

        (* End of Chart: '<S13>/Chart_REQ_MAIN_Precharge' *)
        

        (* SignalConversion: '<S678>/Signal Copy' *)
        rtb_IT_boUDC_SafeToShutdown := IP_boSafeToShutdown;
        (* Sum: '<S674>/Add' incorporates:
         *  ArithShift: '<S673>/Shift Arithmetic'
         *  DataTypeConversion: '<S673>/Data Type Conversion'
         *  Sum: '<S673>/Add' *)
        rtb_Add_kr := UDINT_TO_DINT(DINT_TO_UDINT(DWORD_TO_DINT(SHL(DINT_TO_DWORD(USINT_TO_DINT(C_UDC_Msg1[2])), 8))) + USINT_TO_UDINT(C_UDC_Msg1[1]));
        (* Switch: '<S674>/Switch' *)

        IF C_UDC_Msg1_Timeout THEN 
            (* SignalConversion: '<S678>/Signal Copy3' incorporates:
             *  Constant: '<S665>/SafeValue_NA ' *)
            rtb_Add_kr := 0;
        END_IF;

        (* End of Switch: '<S674>/Switch' *)
        

        (* Outputs for Atomic SubSystem: '<S676>/BatteryPackSignals' *)
        (* Switch: '<S120>/Switch' incorporates:
         *  Constant: '<S120>/Constant'
         *  SignalConversion: '<S682>/BusConversion_InsertedFor_IT_BatterySignal_Databus_at_inport_0' *)

        IF rtb_IP_boBMS_HV_REL_ON_BB1 THEN 
            rtb_Add_ci := rtb_Min;
        ELSE 
            rtb_Add_ci := 0.0;
        END_IF;

        (* End of Switch: '<S120>/Switch' *)
        

        (* Switch: '<S120>/Switch1' incorporates:
         *  Constant: '<S120>/Constant'
         *  SignalConversion: '<S682>/BusConversion_InsertedFor_IT_BatterySignal_Databus_at_inport_0' *)

        IF rtb_IP_boBMS_HV_REL_ON_BB2 THEN 
            rtb_Switch5_bs := rtb_Add_an;
        ELSE 
            rtb_Switch5_bs := 0.0;
        END_IF;

        (* End of Switch: '<S120>/Switch1' *)
        

        (* Switch: '<S120>/Switch2' incorporates:
         *  Constant: '<S120>/Constant'
         *  SignalConversion: '<S682>/BusConversion_InsertedFor_IT_BatterySignal_Databus_at_inport_0' *)

        IF rtb_IP_boBMS_HV_REL_ON_BB3 THEN 
            rtb_FL_sSS_MaxDisChargeCurrent := rtb_Add_e;
        ELSE 
            rtb_FL_sSS_MaxDisChargeCurrent := 0.0;
        END_IF;

        (* End of Switch: '<S120>/Switch2' *)
        (* End of Outputs for SubSystem: '<S676>/BatteryPackSignals' *)
        

        (* MinMax: '<S120>/Min' *)
        b_temp2 := MAX(rtb_Add_ci, rtb_Switch5_bs);
        maxV := MAX(b_temp2, rtb_FL_sSS_MaxDisChargeCurrent);
        (* Logic: '<S7>/NOT' incorporates:
         *  MinMax: '<S120>/Min'
         *  RelationalOperator: '<S14>/Compare'
         *  SignalConversion: '<S678>/Signal Copy'
         *  UnitDelay: '<S13>/Unit Delay5' *)
        i0_Chart_PrechargeStatus(ssMethodType := SS_OUTPUT, REQ_MainHV_ON_Precharge := DO_REQ_MainHV_ON_Precharge, LoadCurrent :=  NOT IP_boSafeToShutdown, LoadVoltage := DINT_TO_REAL(rtb_Add_kr), SystemVoltage := maxV, KL15_CM_diable := rtb_FL_boKL15_Disable, MainHV_Minus_Status := UnitDelay5_DSTATE_e);
        Precharge_Satus := i0_Chart_PrechargeStatus.Precharge_Satus;
        (* Logic: '<S13>/OR' *)
        rtb_Out_bl := (rtb_Delay_j OR rtb_FL_boSS_HVIL_NOK) OR rtb_out_l;
        (* Chart: '<S13>/delay' incorporates:
         *  Constant: '<S13>/Constant1' *)
        (* Gateway: ChiefMaster/Flow Logic/BDU Control/BDUSystem/delay *)
        (* During: ChiefMaster/Flow Logic/BDU Control/BDUSystem/delay *)

        IF is_active_c4_ChiefMaster = 0 THEN 
            (* Entry: ChiefMaster/Flow Logic/BDU Control/BDUSystem/delay *)
            is_active_c4_ChiefMaster := 1;
            (* Entry Internal: ChiefMaster/Flow Logic/BDU Control/BDUSystem/delay *)
            (* Transition: '<S24>:2' *)
            is_c4_ChiefMaster := ChiefMaster_IN_Default_i2;
            (* Entry 'Default': '<S24>:1' *)
            (* '<S24>:1:2' Out = false *)
            rtb_Out_bl := FALSE;
        ELSE 

            CASE is_c4_ChiefMaster OF
                ChiefMaster_IN_Actual_o: 
                    (* During 'Actual': '<S24>:11' *)
                    (* Transition: '<S24>:17' *)
                    (* '<S24>:14:1' sf_internal_predicateOutput = In == false; *)

                    IF  NOT rtb_Out_bl THEN 
                        (* Transition: '<S24>:14' *)
                        is_c4_ChiefMaster := ChiefMaster_IN_Default_i2;
                        (* Entry 'Default': '<S24>:1' *)
                        (* '<S24>:1:2' Out = false *)
                    END_IF;

                ChiefMaster_IN_Default_i2: 
                    (* During 'Default': '<S24>:1' *)
                    (* '<S24>:5:1' sf_internal_predicateOutput = In == true; *)

                    IF rtb_Out_bl THEN 
                        (* Transition: '<S24>:5' *)
                        is_c4_ChiefMaster := ChiefMaster_IN_hold_oa;
                        temporalCounter_i1_m(timerAction := 1, maxTime := 0);
                        (* Entry 'hold': '<S24>:4' *)
                        (* '<S24>:4:2' Out = false *)
                        rtb_Out_bl := FALSE;
                    END_IF;

                ELSE
                    (* During 'hold': '<S24>:4' *)
                    (* '<S24>:12:1' sf_internal_predicateOutput = after(DelayTime_s,sec); *)
                    temporalCounter_i1_m(timerAction := 2, maxTime := TRUNC(REAL_TO_LREAL(MainHV_Minus_In_Delay) * 1000.0));

                    IF temporalCounter_i1_m.done THEN 
                        (* Transition: '<S24>:12' *)
                        is_c4_ChiefMaster := ChiefMaster_IN_Actual_o;
                        (* Entry 'Actual': '<S24>:11' *)
                        (* '<S24>:11:2' Out = In *)
                    ELSE 
                        (* Transition: '<S24>:16' *)
                        (* '<S24>:14:1' sf_internal_predicateOutput = In == false; *)

                        IF  NOT rtb_Out_bl THEN 
                            (* Transition: '<S24>:14' *)
                            is_c4_ChiefMaster := ChiefMaster_IN_Default_i2;
                            (* Entry 'Default': '<S24>:1' *)
                            (* '<S24>:1:2' Out = false *)
                        ELSE 
                            (* '<S24>:4:2' Out = false *)
                            rtb_Out_bl := FALSE;
                        END_IF;

                    END_IF;

            END_CASE;

        END_IF;

        (* End of Chart: '<S13>/delay' *)
        

        (* UnitDelay: '<S13>/Unit Delay1' *)
        rtb_UnitDelay1_d := UnitDelay1_DSTATE_b;
        (* UnitDelay: '<S110>/Unit Delay' *)
        rtb_UnitDelay := UnitDelay_DSTATE_h;
        (* Outputs for Atomic SubSystem: '<S676>/BatteryPackSignals' *)
        (* Switch: '<S110>/Switch3' incorporates:
         *  Constant: '<S110>/Constant1'
         *  Constant: '<S110>/Constant2'
         *  Logic: '<S110>/OR'
         *  SignalConversion: '<S682>/BusConversion_InsertedFor_IT_BatterySignal_Databus_at_inport_0' *)

        IF (rtb_IP_boBMS_HV_REL_ON_BB1 OR rtb_IP_boBMS_HV_REL_ON_BB2) OR rtb_IP_boBMS_HV_REL_ON_BB3 THEN 
            rtb_FL_sSS_MaxDisChargeCurrent := NotAvailable_uint16;
        ELSE 
            rtb_FL_sSS_MaxDisChargeCurrent := 0.0;
        END_IF;

        (* End of Switch: '<S110>/Switch3' *)
        

        (* Switch: '<S110>/Switch' incorporates:
         *  SignalConversion: '<S682>/BusConversion_InsertedFor_IT_BatterySignal_Databus_at_inport_0' *)

        IF rtb_IP_boBMS_HV_REL_ON_BB1 THEN 
            rtb_Switch5_bs := rtb_Add_b;
        ELSE 
            rtb_Switch5_bs := rtb_FL_sSS_MaxDisChargeCurrent;
        END_IF;

        (* End of Switch: '<S110>/Switch' *)
        

        (* Switch: '<S110>/Switch1' incorporates:
         *  SignalConversion: '<S682>/BusConversion_InsertedFor_IT_BatterySignal_Databus_at_inport_0' *)

        IF rtb_IP_boBMS_HV_REL_ON_BB2 THEN 
            rtb_Add_ci := rtb_Add_h;
        ELSE 
            rtb_Add_ci := rtb_FL_sSS_MaxDisChargeCurrent;
        END_IF;

        (* End of Switch: '<S110>/Switch1' *)
        

        (* Switch: '<S110>/Switch2' incorporates:
         *  SignalConversion: '<S682>/BusConversion_InsertedFor_IT_BatterySignal_Databus_at_inport_0' *)

        IF rtb_IP_boBMS_HV_REL_ON_BB3 THEN 
            rtb_Divide_h := rtb_Add_g;
        ELSE 
            rtb_Divide_h := rtb_FL_sSS_MaxDisChargeCurrent;
        END_IF;

        (* End of Switch: '<S110>/Switch2' *)
        

        (* Sum: '<S110>/Add' incorporates:
         *  SignalConversion: '<S682>/BusConversion_InsertedFor_IT_BatterySignal_Databus_at_inport_0'
         *  Sum: '<S121>/Add' *)
        rtb_ExtractDesiredBits_bk_tmp := UDINT_TO_USINT((BOOL_TO_UDINT(rtb_IP_boBMS_HV_REL_ON_BB1) + BOOL_TO_UDINT(rtb_IP_boBMS_HV_REL_ON_BB2)) + BOOL_TO_UDINT(rtb_IP_boBMS_HV_REL_ON_BB3));
        (* End of Outputs for SubSystem: '<S676>/BatteryPackSignals' *)
        

        (* RelationalOperator: '<S190>/Compare' incorporates:
         *  Constant: '<S190>/Constant' *)
        rtb_Switch_b := rtb_ExtractDesiredBits_bk_tmp = 1;
        (* RelationalOperator: '<S191>/Compare' incorporates:
         *  Constant: '<S191>/Constant' *)
        rtb_Switch1_fj := rtb_ExtractDesiredBits_b13 > 0;
        (* Outputs for Atomic SubSystem: '<S676>/BatteryPackSignals' *)
        (* Logic: '<S121>/OR3' incorporates:
         *  Logic: '<S121>/AND'
         *  Logic: '<S121>/AND1'
         *  Logic: '<S121>/AND2'
         *  SignalConversion: '<S682>/BusConversion_InsertedFor_IT_BatterySignal_Databus_at_inport_0'
         *  UnitDelay: '<S121>/Unit Delay'
         *  UnitDelay: '<S121>/Unit Delay1'
         *  UnitDelay: '<S121>/Unit Delay2' *)
        rtb_FL_boSS_BDU_Reset := ((((rtb_IP_boBMS_HV_REL_ON_BB1 AND rtb_Switch_b) AND rtb_Switch1_fj) AND UnitDelay_DSTATE_d) OR (((rtb_Switch1_fj AND rtb_Switch_b) AND rtb_IP_boBMS_HV_REL_ON_BB2) AND UnitDelay1_DSTATE_m)) OR (((rtb_IP_boBMS_HV_REL_ON_BB3 AND rtb_Switch_b) AND rtb_Switch1_fj) AND UnitDelay2_DSTATE_m);
        (* End of Outputs for SubSystem: '<S676>/BatteryPackSignals' *)
        

        (* Logic: '<S55>/NOR' *)
        rtb_FL_boKL15_Reset := (( NOT rtb_IT_boUDC_KL15_D) AND ( NOT rtb_IT_boUDC_KL15_C)) AND rtb_out_n;
        (* End of Outputs for SubSystem: '<Root>/ChiefMaster' *)
        

        (* Constant: '<S388>/Constant4' incorporates:
         *  Constant: '<S388>/Constant'
         *  Constant: '<S388>/Constant1'
         *  Constant: '<S388>/Constant2'
         *  Constant: '<S388>/Constant3' *)
        i0_Chart_Hysteresis_LowActive(ssMethodType := SS_OUTPUT, sSignal := AI_MainHV_Minus_FB, boInitial_Value := FALSE, boValue_Activated := TRUE, boValue_Deactivated := FALSE, sLB := 5000.0, b_sUB := 10000.0);
        boOutput_n := i0_Chart_Hysteresis_LowActive.boOutput;
        (* Constant: '<S382>/Constant4' incorporates:
         *  Constant: '<S382>/Constant'
         *  Constant: '<S382>/Constant1'
         *  Constant: '<S382>/Constant2'
         *  Constant: '<S382>/Constant3' *)
        i0_Chart_Hysteresis_HighActive(ssMethodType := SS_OUTPUT, sSignal := AI_EmergencyButton_NC, boInitial_Value := FALSE, boValue_Activated := TRUE, boValue_Deactivated := FALSE, sLB := 2000.0, b_sUB := 8000.0);
        boOutput_h := i0_Chart_Hysteresis_HighActive.boOutput;
        (* Outputs for Atomic SubSystem: '<Root>/ChiefMaster' *)
        (* SignalConversion: '<S677>/Signal Copy5' *)
        rtb_IT_boHW_MainHV_Minus_FB := boOutput_n;
        (* SignalConversion: '<S677>/Signal Copy6' *)
        rtb_IT_sHW_EmergencyButton_NC := boOutput_h;
        (* End of Outputs for SubSystem: '<Root>/ChiefMaster' *)
        

        (* Constant: '<S383>/Constant4' incorporates:
         *  Constant: '<S383>/Constant'
         *  Constant: '<S383>/Constant1'
         *  Constant: '<S383>/Constant2'
         *  Constant: '<S383>/Constant3' *)
        i1_Chart_Hysteresis_HighActive(ssMethodType := SS_OUTPUT, sSignal := AI_EmergencyButton_NO, boInitial_Value := FALSE, boValue_Activated := TRUE, boValue_Deactivated := FALSE, sLB := 18000.0, b_sUB := 22000.0);
        boOutput_k := i1_Chart_Hysteresis_HighActive.boOutput;
        (* Outputs for Atomic SubSystem: '<Root>/ChiefMaster' *)
        (* SignalConversion: '<S677>/Signal Copy7' *)
        rtb_IT_boHW_EmergencyButton_NO := boOutput_k;
        (* End of Outputs for SubSystem: '<Root>/ChiefMaster' *)
        

        (* Constant: '<S384>/Constant4' incorporates:
         *  Constant: '<S384>/Constant'
         *  Constant: '<S384>/Constant1'
         *  Constant: '<S384>/Constant2'
         *  Constant: '<S384>/Constant3' *)
        i2_Chart_Hysteresis_HighActive(ssMethodType := SS_OUTPUT, sSignal := AI_HVIL_BDU, boInitial_Value := FALSE, boValue_Activated := TRUE, boValue_Deactivated := FALSE, sLB := 12000.0, b_sUB := 15000.0);
        boOutput_l := i2_Chart_Hysteresis_HighActive.boOutput;
        (* Constant: '<S384>/Constant5' *)
        i0_HVIL_Input_Delay(ssMethodType := SS_OUTPUT, HVIL_IN := boOutput_l, IP_HVIL_Delay_ms := IP_u8HVIL_Delay_ms);
        rtb_out_l := i0_HVIL_Input_Delay.out;
        (* Constant: '<S385>/Constant4' incorporates:
         *  Constant: '<S385>/Constant'
         *  Constant: '<S385>/Constant1'
         *  Constant: '<S385>/Constant2'
         *  Constant: '<S385>/Constant3' *)
        i3_Chart_Hysteresis_HighActive(ssMethodType := SS_OUTPUT, sSignal := AI_HVIL_Component, boInitial_Value := FALSE, boValue_Activated := TRUE, boValue_Deactivated := FALSE, sLB := 12000.0, b_sUB := 15000.0);
        boOutput_p := i3_Chart_Hysteresis_HighActive.boOutput;
        (* Constant: '<S385>/Constant5' *)
        i1_HVIL_Input_Delay(ssMethodType := SS_OUTPUT, HVIL_IN := boOutput_p, IP_HVIL_Delay_ms := IP_u8HVIL_Delay_ms);
        rtb_FL_boHVC_AllCellBalanced := i1_HVIL_Input_Delay.out;
        (* Constant: '<S386>/Constant4' incorporates:
         *  Constant: '<S386>/Constant'
         *  Constant: '<S386>/Constant1'
         *  Constant: '<S386>/Constant2'
         *  Constant: '<S386>/Constant3' *)
        i4_Chart_Hysteresis_HighActive(ssMethodType := SS_OUTPUT, sSignal := AI_HVIL_Battery, boInitial_Value := FALSE, boValue_Activated := TRUE, boValue_Deactivated := FALSE, sLB := 12000.0, b_sUB := 15000.0);
        boOutput_f := i4_Chart_Hysteresis_HighActive.boOutput;
        (* Constant: '<S386>/Constant5' *)
        i2_HVIL_Input_Delay(ssMethodType := SS_OUTPUT, HVIL_IN := boOutput_f, IP_HVIL_Delay_ms := IP_u8HVIL_Delay_ms);
        rtb_out_n := i2_HVIL_Input_Delay.out;
        (* Outputs for Atomic SubSystem: '<Root>/ChiefMaster' *)
        (* SignalConversion: '<S677>/Signal Copy8' *)
        i3_Chart_SetDominantSwitch(ssMethodType := SS_OUTPUT, boData_In := DI_ResetButton_LED_NO, boReset := rtb_FL_boKL15_Reset);
        rtb_boData_Out := i3_Chart_SetDominantSwitch.boData_Out;
        (* SignalConversion: '<S677>/Signal Copy1' incorporates:
         *  SignalConversion: '<S677>/Signal Copy14'
         *  SignalConversion: '<S677>/Signal Copy2'
         *  SignalConversion: '<S677>/Signal Copy3' *)
        i0_EmergencySD(ssMethodType := SS_OUTPUT, FL_boKL15_Reset := rtb_FL_boKL15_Reset, IT_boEmergencySwitch_NC := rtb_IT_sHW_EmergencyButton_NC, IT_boEmergencySwitch_NO := rtb_IT_boHW_EmergencyButton_NO, IT_boHW_HVIL_BDU := rtb_out_l, IT_boHW_HVIL_Components := rtb_FL_boHVC_AllCellBalanced, IT_boHW_HVIL_Battery := rtb_out_n, IT_boHW_HVIL_Overrule := DI_HVIL_Overrule, IT_boHW_ResetButton_LED_NO_State := rtb_boData_Out);
        rtb_Delay_j := i0_EmergencySD.FL_boSS_System_ESD;
        rtb_Out := i0_EmergencySD.FL_u8SS_EmergencyStopState;
        rtb_FL_boSS_HVIL_NOK := i0_EmergencySD.FL_boHVIL_NOK;
        (* Constant: '<S392>/Constant' *)
        b_Constant := USINT_TO_UINT(IP_u8HW_IN_delay_ms);
        (* End of Outputs for SubSystem: '<Root>/ChiefMaster' *)
        i0_Input_Delay(ssMethodType := SS_OUTPUT, IP_u8HW_IN_delay_ms_m := b_Constant, Input := DI_Proximity_BB1);
        rtb_IT_boHW_HVIL_BDU := i0_Input_Delay.out;
        (* Outputs for Atomic SubSystem: '<Root>/ChiefMaster' *)
        (* Constant: '<S393>/Constant' *)
        Constant_n := USINT_TO_UINT(IP_u8HW_IN_delay_ms);
        (* End of Outputs for SubSystem: '<Root>/ChiefMaster' *)
        i1_Input_Delay(ssMethodType := SS_OUTPUT, IP_u8HW_IN_delay_ms_m := Constant_n, Input := DI_Proximity_BB2);
        rtb_out_i := i1_Input_Delay.out;
        (* Outputs for Atomic SubSystem: '<Root>/ChiefMaster' *)
        (* Constant: '<S394>/Constant' *)
        Constant_o := USINT_TO_UINT(IP_u8HW_IN_delay_ms);
        (* End of Outputs for SubSystem: '<Root>/ChiefMaster' *)
        i2_Input_Delay(ssMethodType := SS_OUTPUT, IP_u8HW_IN_delay_ms_m := Constant_o, Input := DI_Proximity_BB3);
        rtb_out_ne := i2_Input_Delay.out;
        (* Outputs for Atomic SubSystem: '<Root>/ChiefMaster' *)
        (* Outputs for Atomic SubSystem: '<S676>/BatteryPackSignals' *)
        (* SignalConversion: '<S682>/BusConversion_InsertedFor_IT_BatterySignal_Databus_at_inport_0' incorporates:
         *  SignalConversion: '<S677>/Signal Copy10'
         *  SignalConversion: '<S677>/Signal Copy11'
         *  SignalConversion: '<S677>/Signal Copy9'
         *  SignalConversion: '<S698>/Signal Copy'
         *  SignalConversion: '<S699>/Signal Copy'
         *  SignalConversion: '<S700>/Signal Copy' *)
        i0_SDError(ssMethodType := SS_OUTPUT, FL_boKL15_Reset := rtb_FL_boKL15_Reset, IT_Databus := rtb_ExtractDesiredBits_b13, IT_Databus_m := rtb_IP_boBMS_HV_REL_ON_BB1, IT_Databus_n := rtb_IP_boBMS_SDError_BB1, IT_Databus_a := rtb_IP_boBMS_HV_REL_ON_BB2, IT_Databus_o := rtb_IP_boBMS_SDError_BB2, IT_Databus_or := rtb_IP_boBMS_HV_REL_ON_BB3, IT_Databus_i := rtb_IP_boBMS_SDError_BB3, IT_Databus_c := rtb_Add_ki5, IT_Databus_o3 := rtb_Add_ir, IT_Databus_e := rtb_Add_m, IT_Databus_n0 := rtb_IT_boHW_HVIL_BDU, IT_Databus_ep := rtb_out_i, IT_Databus_l := rtb_out_ne, IT_Databus_f := rtb_IP_boBMS_IMD_Active_BB1, IT_Databus_k := rtb_IP_boBMS_IMD_Active_BB2, IT_Databus_g := rtb_IP_boBMS_IMD_Active_BB3, IT_Databus_b := rtb_S_in, IT_Databus_d := rtb_AND_l2, IT_Databus_h := rtb_IP_boBatt1_Actia_Availability, IT_Databus_j := rtb_AND_ni, IT_Databus_ja := rtb_Delay_dl, IT_Databus_if := rtb_AND_ma, FL_BDUControl_Databus := MainHV_Minus_Status, FL_BDUControl_Databus_o := MainHV_Plus_Status, FL_BDUControl_Databus_n := Precharge_Satus, FL_BatteryBox_HVControl_Databus := REQ_HV_ON_a, FL_BatteryBox_HVControl_Databus_b := REQ_HV_ON_d, FL_BatteryBox_HVControl_Databus_a := REQ_HV_ON, FL_u8SS_EmergencySD := rtb_Delay_j);
        System_Error := i0_SDError.FL_boSS_System_SD;
        rtb_System_SD_ErrorCode := i0_SDError.FL_u8SS_System_SD_ErrorCode;
        (* Switch: '<S117>/Switch' incorporates:
         *  Constant: '<S117>/Constant'
         *  SignalConversion: '<S682>/BusConversion_InsertedFor_IT_BatterySignal_Databus_at_inport_0'
         *  SignalConversion: '<S698>/Signal Copy' *)

        IF rtb_IP_boBMS_HV_REL_ON_BB1 THEN 
            rtb_Switch_b := rtb_IP_boBMS_SDError_BB1;
        ELSE 
            rtb_Switch_b := FALSE;
        END_IF;

        (* End of Switch: '<S117>/Switch' *)
        

        (* Switch: '<S117>/Switch1' incorporates:
         *  Constant: '<S117>/Constant'
         *  SignalConversion: '<S682>/BusConversion_InsertedFor_IT_BatterySignal_Databus_at_inport_0'
         *  SignalConversion: '<S699>/Signal Copy' *)

        IF rtb_IP_boBMS_HV_REL_ON_BB2 THEN 
            rtb_Switch1_fj := rtb_IP_boBMS_SDError_BB2;
        ELSE 
            rtb_Switch1_fj := FALSE;
        END_IF;

        (* End of Switch: '<S117>/Switch1' *)
        

        (* Switch: '<S117>/Switch2' incorporates:
         *  Constant: '<S117>/Constant'
         *  SignalConversion: '<S682>/BusConversion_InsertedFor_IT_BatterySignal_Databus_at_inport_0'
         *  SignalConversion: '<S700>/Signal Copy' *)

        IF rtb_IP_boBMS_HV_REL_ON_BB3 THEN 
            rtb_Switch2_d := rtb_IP_boBMS_SDError_BB3;
        ELSE 
            rtb_Switch2_d := FALSE;
        END_IF;

        (* End of Switch: '<S117>/Switch2' *)
        (* End of Outputs for SubSystem: '<S676>/BatteryPackSignals' *)
        

        (* Logic: '<S117>/OR' *)
        rtb_FL_boSS_System_Error := (rtb_Switch_b OR rtb_Switch1_fj) OR rtb_Switch2_d;
        (* Switch: '<S110>/Switch7' incorporates:
         *  Constant: '<S110>/Constant3'
         *  Constant: '<S110>/Constant4' *)

        IF UnexpectedBattChargingFcn_Available THEN 
            rtb_Uk1 := 0.0;
        ELSE 
            rtb_Uk1 := PLC_BOOL_TO_LREAL(in := rtb_FL_boKL15_Disable);
        END_IF;

        (* End of Switch: '<S110>/Switch7' *)
        

        (* Logic: '<S110>/NOT' incorporates:
         *  Logic: '<S110>/NOR1'
         *  Logic: '<S110>/OR2' *)
        rtb_NOT_m5 := (( NOT rtb_FL_boSS_BDU_Reset) AND ((( NOT rtb_Delay_j) AND ( NOT System_Error)) AND ( NOT rtb_FL_boSS_System_Error))) AND (rtb_Uk1 = 0.0);
        (* Outputs for Atomic SubSystem: '<S676>/BatteryPackSignals' *)
        (* Switch: '<S128>/Switch' incorporates:
         *  Constant: '<S128>/Constant'
         *  SignalConversion: '<S682>/BusConversion_InsertedFor_IT_BatterySignal_Databus_at_inport_0' *)

        IF rtb_IP_boBMS_HV_REL_ON_BB1 THEN 
            rtb_Uk1 := REAL_TO_LREAL(rtb_Add_ki5);
        ELSE 
            rtb_Uk1 := 65535.0;
        END_IF;

        (* End of Switch: '<S128>/Switch' *)
        

        (* Switch: '<S128>/Switch1' incorporates:
         *  Constant: '<S128>/Constant1'
         *  SignalConversion: '<S682>/BusConversion_InsertedFor_IT_BatterySignal_Databus_at_inport_0' *)

        IF rtb_IP_boBMS_HV_REL_ON_BB2 THEN 
            rtb_UnitDelay2 := REAL_TO_LREAL(rtb_Add_ir);
        ELSE 
            rtb_UnitDelay2 := 65535.0;
        END_IF;

        (* End of Switch: '<S128>/Switch1' *)
        

        (* Switch: '<S128>/Switch2' incorporates:
         *  Constant: '<S128>/Constant2'
         *  SignalConversion: '<S682>/BusConversion_InsertedFor_IT_BatterySignal_Databus_at_inport_0' *)

